LIN {X 0,Y 136.001,Z 403.544,A -85,B 0,C 180,E1 -24793.658,E2 -24793.658} C_VEL
LIN {X 0,Y 136.034,Z 403.535,A -85,B 0,C 180,E1 -24797.807,E2 -24797.807} C_VEL
LIN {X 0,Y 136.073,Z 403.535,A -85,B 0,C 180,E1 -24801.699,E2 -24801.699} C_VEL
LIN {X 0,Y 136.278,Z 403.501,A -85,B 0,C 180,E1 -24805.603,E2 -24805.603} C_VEL
LIN {X 0,Y 136.386,Z 403.498,A -85,B 0,C 180,E1 -24808.982,E2 -24808.982} C_VEL
LIN {X 0,Y 136.062,Z 403.665,A -85,B 0,C 180,E1 -24810.402,E2 -24810.402} C_VEL
LIN {X 0,Y 135.119,Z 409.074,A -85,B 0,C 180,E1 -24817.039,E2 -24817.039} C_VEL
LIN {X 0,Y 134.458,Z 414.255,A -85,B 0,C 180,E1 -24823.293,E2 -24823.293} C_VEL
LIN {X 0,Y 135.285,Z 420.732,A -85,B 0,C 180,E1 -24831.034,E2 -24831.034} C_VEL
LIN {X 0,Y 135.533,Z 421.149,A -85,B 0,C 180,E1 -24831.52,E2 -24831.52} C_VEL
LIN {X 0,Y 136.845,Z 432.369,A -85,B 0,C 180,E1 -24833.364,E2 -24833.364} C_VEL
LIN {X 0,Y 136.477,Z 444.992,A -85,B 0,C 180,E1 -24836.309,E2 -24836.309} C_VEL
LIN {X 0,Y 136.219,Z 455.03,A -85,B 0,C 180,E1 -24839.261,E2 -24839.261} C_VEL
LIN {X 0,Y 136.014,Z 464.96,A -85,B 0,C 180,E1 -24842.962,E2 -24842.962} C_VEL
LIN {X 0,Y 136.62,Z 474.818,A -85,B 0,C 180,E1 -24847.389,E2 -24847.389} C_VEL
LIN {X 0,Y 138.11,Z 482.79,A -85,B 0,C 180,E1 -24851.744,E2 -24851.744} C_VEL
LIN {X 0,Y 140.744,Z 489.39,A -85,B 0,C 180,E1 -24855.941,E2 -24855.941} C_VEL
LIN {X 0,Y 144.372,Z 494.762,A -85,B 0,C 180,E1 -24859.923,E2 -24859.923} C_VEL
LIN {X 0,Y 148.92,Z 499.026,A -85,B 0,C 180,E1 -24863.65,E2 -24863.65} C_VEL
LIN {X 0,Y 154.307,Z 502.234,A -85,B 0,C 180,E1 -24867.094,E2 -24867.094} C_VEL
LIN {X 0,Y 158.302,Z 503.827,A -85,B 0,C 180,E1 -24869.233,E2 -24869.233} C_VEL
LIN {X 0,Y 162.598,Z 504.999,A -85,B 0,C 180,E1 -24871.244,E2 -24871.244} C_VEL
LIN {X 0,Y 169.94,Z 505.976,A -85,B 0,C 180,E1 -24874.196,E2 -24874.196} C_VEL
LIN {X 0,Y 171.965,Z 506.075,A -85,B 0,C 180,E1 -24874.901,E2 -24874.901} C_VEL
LIN {X 0,Y 176.179,Z 506.156,A -85,B 0,C 180,E1 -24876.753,E2 -24876.753} C_VEL
LIN {X 0,Y 178.352,Z 506.601,A -85,B 0,C 180,E1 -24879.086,E2 -24879.086} C_VEL
LIN {X 0,Y 180.016,Z 507.386,A -85,B 0,C 180,E1 -24882.116,E2 -24882.116} C_VEL
LIN {X 0,Y 179.621,Z 508.08,A -85,B 0,C 180,E1 -24883.626,E2 -24883.626} C_VEL
LIN {X 0,Y 177.585,Z 508.851,A -85,B 0,C 180,E1 -24884.572,E2 -24884.572} C_VEL
LIN {X 0,Y 167.712,Z 511.361,A -85,B 0,C 180,E1 -24887.895,E2 -24887.895} C_VEL
LIN {X 0,Y 163.054,Z 512.165,A -85,B 0,C 180,E1 -24889.718,E2 -24889.718} C_VEL
LIN {X 0,Y 154.89,Z 513.005,A -85,B 0,C 180,E1 -24893.852,E2 -24893.852} C_VEL
LIN {X 0,Y 147.172,Z 512.738,A -85,B 0,C 180,E1 -24899.268,E2 -24899.268} C_VEL
LIN {X 0,Y 142.861,Z 511.656,A -85,B 0,C 180,E1 -24903.72,E2 -24903.72} C_VEL
LIN {X 0,Y 139.41,Z 509.457,A -85,B 0,C 180,E1 -24909.335,E2 -24909.335} C_VEL
LIN {X 0,Y 137.831,Z 505.899,A -85,B 0,C 180,E1 -24915.653,E2 -24915.653} C_VEL
LIN {X 0,Y 138.323,Z 501.685,A -85,B 0,C 180,E1 -24921.232,E2 -24921.232} C_VEL
LIN {X 0,Y 139.606,Z 497.302,A -85,B 0,C 180,E1 -24925.669,E2 -24925.669} C_VEL
LIN {X 0,Y 140.175,Z 494.465,A -85,B 0,C 180,E1 -24927.844,E2 -24927.844} C_VEL
LIN {X 0,Y 140.099,Z 489.468,A -85,B 0,C 180,E1 -24930.718,E2 -24930.718} C_VEL
LIN {X 0,Y 139.615,Z 481.506,A -85,B 0,C 180,E1 -24934.33,E2 -24934.33} C_VEL
LIN {X 0,Y 139.3,Z 472.487,A -85,B 0,C 180,E1 -24937.61,E2 -24937.61} C_VEL
LIN {X 0,Y 139.429,Z 464.069,A -85,B 0,C 180,E1 -24940.161,E2 -24940.161} C_VEL
LIN {X 0,Y 137.814,Z 452.885,A -85,B 0,C 180,E1 -24942.565,E2 -24942.565} C_VEL
LIN {X 0,Y 136.785,Z 440.476,A -85,B 0,C 180,E1 -24944.679,E2 -24944.679} C_VEL
LIN {X 0,Y 136.596,Z 432.577,A -85,B 0,C 180,E1 -24945.766,E2 -24945.766} C_VEL
LIN {X 0,Y 136.082,Z 427.218,A -85,B 0,C 180,E1 -24951.193,E2 -24951.193} C_VEL
LIN {X 0,Y 138.905,Z 417.791,A -85,B 0,C 180,E1 -24960.669,E2 -24960.669} C_VEL
LIN {X 0,Y 139.445,Z 416.478,A -85,B 0,C 180,E1 -24961.949,E2 -24961.949} C_VEL
LIN {X 0,Y 138.943,Z 413.586,A -85,B 0,C 180,E1 -24964.73,E2 -24964.73} C_VEL
LIN {X 0,Y 137.461,Z 408.348,A -85,B 0,C 180,E1 -24969.923,E2 -24969.923} C_VEL
LIN {X 0,Y 136.332,Z 403.499,A -85,B 0,C 180,E1 -24975.017,E2 -24975.017} C_VEL
LIN {X 0,Y 136.064,Z 403.536,A -85,B 0,C 180,E1 -24981.697,E2 -24981.697} C_VEL
LIN {X 0,Y 136.09,Z 403.527,A -85,B 0,C 180,E1 -24985.717,E2 -24985.717} C_VEL
LIN {X 0,Y 136.146,Z 403.523,A -85,B 0,C 180,E1 -24992.316,E2 -24992.316} C_VEL
LIN {X 0,Y 136.19,Z 403.52,A -85,B 0,C 180,E1 -24998.168,E2 -24998.168} C_VEL
LIN {X 0,Y 135.722,Z 403.592,A -85,B 0,C 180,E1 -25000.636,E2 -25000.636} C_VEL
LIN {X 0,Y 134.282,Z 403.775,A -85,B 0,C 180,E1 -25003.077,E2 -25003.077} C_VEL
LIN {X 0,Y 129.836,Z 404.308,A -85,B 0,C 180,E1 -25009.8,E2 -25009.8} C_VEL
LIN {X 0,Y 129.486,Z 404.346,A -85,B 0,C 180,E1 -25011.576,E2 -25011.576} C_VEL
LIN {X 0,Y 130.091,Z 404.274,A -85,B 0,C 180,E1 -25020,E2 -25020} C_VEL
LIN {X 0,Y 129.531,Z 404.344,A -85,B 0,C 180,E1 -25029.368,E2 -25029.368} C_VEL
LIN {X 0,Y 129.395,Z 404.366,A -85,B 0,C 180,E1 -25032.548,E2 -25032.548} C_VEL
LIN {X 0,Y 129.164,Z 404.393,A -85,B 0,C 180,E1 -25039.055,E2 -25039.055} C_VEL
LIN {X 0,Y 129.109,Z 404.402,A -85,B 0,C 180,E1 -25042.398,E2 -25042.398} C_VEL
LIN {X 0,Y 129.036,Z 404.412,A -85,B 0,C 180,E1 -25049.374,E2 -25049.374} C_VEL
LIN {X 0,Y 128.961,Z 404.416,A -85,B 0,C 180,E1 -25055.17,E2 -25055.17} C_VEL
LIN {X 0,Y 128.934,Z 404.422,A -85,B 0,C 180,E1 -25060.852,E2 -25060.852} C_VEL
LIN {X 0,Y 128.922,Z 404.425,A -85,B 0,C 180,E1 -25065.128,E2 -25065.128} C_VEL
LIN {X 0,Y 128.958,Z 404.418,A -85,B 0,C 180,E1 -25069.728,E2 -25069.728} C_VEL
LIN {X 0,Y 128.993,Z 404.418,A -85,B 0,C 180,E1 -25074.811,E2 -25074.811} C_VEL
LIN {X 0,Y 129.034,Z 404.406,A -85,B 0,C 180,E1 -25080.647,E2 -25080.647} C_VEL
LIN {X 0,Y 129.137,Z 404.395,A -85,B 0,C 180,E1 -25087.607,E2 -25087.607} C_VEL
LIN {X 0,Y 129.188,Z 404.391,A -85,B 0,C 180,E1 -25090.95,E2 -25090.95} C_VEL
LIN {X 0,Y 129.418,Z 404.357,A -85,B 0,C 180,E1 -25097.821,E2 -25097.821} C_VEL
LIN {X 0,Y 129.519,Z 404.351,A -85,B 0,C 180,E1 -25100.632,E2 -25100.632} C_VEL
LIN {X 0,Y 130.092,Z 404.281,A -85,B 0,C 180,E1 -25110.001,E2 -25110.001} C_VEL
LIN {X 0,Y 129.479,Z 404.356,A -85,B 0,C 180,E1 -25119.372,E2 -25119.372} C_VEL
LIN {X 0,Y 129.347,Z 404.365,A -85,B 0,C 180,E1 -25122.553,E2 -25122.553} C_VEL
LIN {X 0,Y 129.159,Z 404.395,A -85,B 0,C 180,E1 -25129.056,E2 -25129.056} C_VEL
LIN {X 0,Y 129.111,Z 404.398,A -85,B 0,C 180,E1 -25132.399,E2 -25132.399} C_VEL
LIN {X 0,Y 129.038,Z 404.406,A -85,B 0,C 180,E1 -25139.374,E2 -25139.374} C_VEL
LIN {X 0,Y 128.995,Z 404.418,A -85,B 0,C 180,E1 -25145.19,E2 -25145.19} C_VEL
LIN {X 0,Y 128.953,Z 404.419,A -85,B 0,C 180,E1 -25150.845,E2 -25150.845} C_VEL
LIN {X 0,Y 128.924,Z 404.423,A -85,B 0,C 180,E1 -25155.128,E2 -25155.128} C_VEL
LIN {X 0,Y 128.987,Z 404.417,A -85,B 0,C 180,E1 -25159.713,E2 -25159.713} C_VEL
LIN {X 0,Y 129.144,Z 404.393,A -85,B 0,C 180,E1 -25164.717,E2 -25164.717} C_VEL
LIN {X 0,Y 129.235,Z 404.374,A -85,B 0,C 180,E1 -25167.056,E2 -25167.056} C_VEL
LIN {X 0,Y 128.884,Z 404.599,A -85,B 0,C 180,E1 -25171.009,E2 -25171.009} C_VEL
LIN {X 0,Y 127.961,Z 409.6,A -85,B 0,C 180,E1 -25177.39,E2 -25177.39} C_VEL
LIN {X 0,Y 127.313,Z 414.748,A -85,B 0,C 180,E1 -25183.977,E2 -25183.977} C_VEL
LIN {X 0,Y 128.098,Z 420.318,A -85,B 0,C 180,E1 -25190.957,E2 -25190.957} C_VEL
LIN {X 0,Y 128.762,Z 421.528,A -85,B 0,C 180,E1 -25192.435,E2 -25192.435} C_VEL
LIN {X 0,Y 130.011,Z 431.845,A -85,B 0,C 180,E1 -25194.183,E2 -25194.183} C_VEL
LIN {X 0,Y 129.718,Z 443.147,A -85,B 0,C 180,E1 -25196.894,E2 -25196.894} C_VEL
LIN {X 0,Y 129.538,Z 453.363,A -85,B 0,C 180,E1 -25200,E2 -25200} C_VEL
LIN {X 0,Y 129.381,Z 463.671,A -85,B 0,C 180,E1 -25203.893,E2 -25203.893} C_VEL
LIN {X 0,Y 129.901,Z 472.26,A -85,B 0,C 180,E1 -25207.773,E2 -25207.773} C_VEL
LIN {X 0,Y 131.762,Z 482.01,A -85,B 0,C 180,E1 -25213.102,E2 -25213.102} C_VEL
LIN {X 0,Y 134.607,Z 488.854,A -85,B 0,C 180,E1 -25217.47,E2 -25217.47} C_VEL
LIN {X 0,Y 139.21,Z 495.266,A -85,B 0,C 180,E1 -25222.249,E2 -25222.249} C_VEL
LIN {X 0,Y 144.183,Z 499.613,A -85,B 0,C 180,E1 -25226.021,E2 -25226.021} C_VEL
LIN {X 0,Y 147.992,Z 501.924,A -85,B 0,C 180,E1 -25228.352,E2 -25228.352} C_VEL
LIN {X 0,Y 152.112,Z 503.822,A -85,B 0,C 180,E1 -25230.546,E2 -25230.546} C_VEL
LIN {X 0,Y 156.554,Z 505.286,A -85,B 0,C 180,E1 -25232.595,E2 -25232.595} C_VEL
LIN {X 0,Y 164.524,Z 506.798,A -85,B 0,C 180,E1 -25235.744,E2 -25235.744} C_VEL
LIN {X 0,Y 166.167,Z 506.978,A -85,B 0,C 180,E1 -25236.308,E2 -25236.308} C_VEL
LIN {X 0,Y 170.317,Z 507.393,A -85,B 0,C 180,E1 -25238.241,E2 -25238.241} C_VEL
LIN {X 0,Y 172.203,Z 508.123,A -85,B 0,C 180,E1 -25240.768,E2 -25240.768} C_VEL
LIN {X 0,Y 172.597,Z 508.889,A -85,B 0,C 180,E1 -25242.865,E2 -25242.865} C_VEL
LIN {X 0,Y 162.539,Z 510.833,A -85,B 0,C 180,E1 -25246.225,E2 -25246.225} C_VEL
LIN {X 0,Y 157.737,Z 511.376,A -85,B 0,C 180,E1 -25248.061,E2 -25248.061} C_VEL
LIN {X 0,Y 149.294,Z 511.755,A -85,B 0,C 180,E1 -25252.267,E2 -25252.267} C_VEL
LIN {X 0,Y 141.83,Z 511.081,A -85,B 0,C 180,E1 -25257.394,E2 -25257.394} C_VEL
LIN {X 0,Y 136.776,Z 509.594,A -85,B 0,C 180,E1 -25262.454,E2 -25262.454} C_VEL
LIN {X 0,Y 133.152,Z 507.034,A -85,B 0,C 180,E1 -25268.316,E2 -25268.316} C_VEL
LIN {X 0,Y 131.562,Z 503.393,A -85,B 0,C 180,E1 -25274.508,E2 -25274.508} C_VEL
LIN {X 0,Y 131.998,Z 498.616,A -85,B 0,C 180,E1 -25280.808,E2 -25280.808} C_VEL
LIN {X 0,Y 133.399,Z 493.899,A -85,B 0,C 180,E1 -25285.468,E2 -25285.468} C_VEL
LIN {X 0,Y 133.899,Z 490.875,A -85,B 0,C 180,E1 -25287.743,E2 -25287.743} C_VEL
LIN {X 0,Y 133.538,Z 485.851,A -85,B 0,C 180,E1 -25290.525,E2 -25290.525} C_VEL
LIN {X 0,Y 133.112,Z 478.587,A -85,B 0,C 180,E1 -25293.784,E2 -25293.784} C_VEL
LIN {X 0,Y 132.773,Z 469.166,A -85,B 0,C 180,E1 -25297.221,E2 -25297.221} C_VEL
LIN {X 0,Y 132.831,Z 462.944,A -85,B 0,C 180,E1 -25299.133,E2 -25299.133} C_VEL
LIN {X 0,Y 131.036,Z 450.859,A -85,B 0,C 180,E1 -25301.799,E2 -25301.799} C_VEL
LIN {X 0,Y 130.027,Z 438.226,A -85,B 0,C 180,E1 -25304.003,E2 -25304.003} C_VEL
LIN {X 0,Y 129.763,Z 432.188,A -85,B 0,C 180,E1 -25304.932,E2 -25304.932} C_VEL
LIN {X 0,Y 128.957,Z 428.337,A -85,B 0,C 180,E1 -25309.086,E2 -25309.086} C_VEL
LIN {X 0,Y 132.142,Z 416.641,A -85,B 0,C 180,E1 -25321.683,E2 -25321.683} C_VEL
LIN {X 0,Y 132.309,Z 416.249,A -85,B 0,C 180,E1 -25322.085,E2 -25322.085} C_VEL
LIN {X 0,Y 131.69,Z 413.387,A -85,B 0,C 180,E1 -25325.008,E2 -25325.008} C_VEL
LIN {X 0,Y 130.12,Z 407.807,A -85,B 0,C 180,E1 -25330.872,E2 -25330.872} C_VEL
LIN {X 0,Y 129.313,Z 404.374,A -85,B 0,C 180,E1 -25334.799,E2 -25334.799} C_VEL
LIN {X 0,Y 129.005,Z 404.414,A -85,B 0,C 180,E1 -25339.702,E2 -25339.702} C_VEL
LIN {X 0,Y 128.993,Z 404.411,A -85,B 0,C 180,E1 -25344.81,E2 -25344.81} C_VEL
LIN {X 0,Y 129.033,Z 404.411,A -85,B 0,C 180,E1 -25350.646,E2 -25350.646} C_VEL
LIN {X 0,Y 129.108,Z 404.402,A -85,B 0,C 180,E1 -25357.602,E2 -25357.602} C_VEL
LIN {X 0,Y 129.16,Z 404.394,A -85,B 0,C 180,E1 -25360.945,E2 -25360.945} C_VEL
LIN {X 0,Y 129.419,Z 404.364,A -85,B 0,C 180,E1 -25367.815,E2 -25367.815} C_VEL
LIN {X 0,Y 129.486,Z 404.346,A -85,B 0,C 180,E1 -25371.576,E2 -25371.576} C_VEL
LIN {X 0,Y 128.783,Z 404.442,A -85,B 0,C 180,E1 -25374.182,E2 -25374.182} C_VEL
LIN {X 0,Y 127.224,Z 404.637,A -85,B 0,C 180,E1 -25376.756,E2 -25376.756} C_VEL
LIN {X 0,Y 122.783,Z 405.191,A -85,B 0,C 180,E1 -25383.868,E2 -25383.868} C_VEL
LIN {X 0,Y 122.457,Z 405.224,A -85,B 0,C 180,E1 -25385.748,E2 -25385.748} C_VEL
LIN {X 0,Y 122.457,Z 405.228,A -85,B 0,C 180,E1 -25389.914,E2 -25389.914} C_VEL
LIN {X 0,Y 122.287,Z 405.253,A -85,B 0,C 180,E1 -25393.29,E2 -25393.29} C_VEL
LIN {X 0,Y 122.052,Z 405.28,A -85,B 0,C 180,E1 -25400.212,E2 -25400.212} C_VEL
LIN {X 0,Y 121.984,Z 405.287,A -85,B 0,C 180,E1 -25403.785,E2 -25403.785} C_VEL
LIN {X 0,Y 121.939,Z 405.295,A -85,B 0,C 180,E1 -25410.172,E2 -25410.172} C_VEL
LIN {X 0,Y 121.886,Z 405.299,A -85,B 0,C 180,E1 -25416.173,E2 -25416.173} C_VEL
LIN {X 0,Y 121.873,Z 405.299,A -85,B 0,C 180,E1 -25421.439,E2 -25421.439} C_VEL
LIN {X 0,Y 121.885,Z 405.302,A -85,B 0,C 180,E1 -25428.556,E2 -25428.556} C_VEL
LIN {X 0,Y 121.946,Z 405.296,A -85,B 0,C 180,E1 -25434.809,E2 -25434.809} C_VEL
LIN {X 0,Y 121.943,Z 405.289,A -85,B 0,C 180,E1 -25439.827,E2 -25439.827} C_VEL
LIN {X 0,Y 122.069,Z 405.275,A -85,B 0,C 180,E1 -25447.1,E2 -25447.1} C_VEL
LIN {X 0,Y 122.133,Z 405.271,A -85,B 0,C 180,E1 -25453.279,E2 -25453.279} C_VEL
LIN {X 0,Y 122.365,Z 405.235,A -85,B 0,C 180,E1 -25457.527,E2 -25457.527} C_VEL
LIN {X 0,Y 122.448,Z 405.231,A -85,B 0,C 180,E1 -25460.086,E2 -25460.086} C_VEL
LIN {X 0,Y 122.608,Z 405.208,A -85,B 0,C 180,E1 -25466.715,E2 -25466.715} C_VEL
LIN {X 0,Y 123.045,Z 405.159,A -85,B 0,C 180,E1 -25470.001,E2 -25470.001} C_VEL
LIN {X 0,Y 122.428,Z 405.233,A -85,B 0,C 180,E1 -25476.593,E2 -25476.593} C_VEL
LIN {X 0,Y 122.32,Z 405.241,A -85,B 0,C 180,E1 -25482.377,E2 -25482.377} C_VEL
LIN {X 0,Y 122.114,Z 405.273,A -85,B 0,C 180,E1 -25486.725,E2 -25486.725} C_VEL
LIN {X 0,Y 122.026,Z 405.28,A -85,B 0,C 180,E1 -25492.852,E2 -25492.852} C_VEL
LIN {X 0,Y 121.952,Z 405.293,A -85,B 0,C 180,E1 -25497.455,E2 -25497.455} C_VEL
LIN {X 0,Y 121.914,Z 405.294,A -85,B 0,C 180,E1 -25501.254,E2 -25501.254} C_VEL
LIN {X 0,Y 121.914,Z 405.296,A -85,B 0,C 180,E1 -25506.19,E2 -25506.19} C_VEL
LIN {X 0,Y 121.886,Z 405.302,A -85,B 0,C 180,E1 -25511.445,E2 -25511.445} C_VEL
LIN {X 0,Y 121.905,Z 405.295,A -85,B 0,C 180,E1 -25518.545,E2 -25518.545} C_VEL
LIN {X 0,Y 122.098,Z 405.27,A -85,B 0,C 180,E1 -25524.858,E2 -25524.858} C_VEL
LIN {X 0,Y 121.921,Z 405.299,A -85,B 0,C 180,E1 -25529.846,E2 -25529.846} C_VEL
LIN {X 0,Y 121.709,Z 405.375,A -85,B 0,C 180,E1 -25531.483,E2 -25531.483} C_VEL
LIN {X 0,Y 120.729,Z 410.686,A -85,B 0,C 180,E1 -25538.657,E2 -25538.657} C_VEL
LIN {X 0,Y 120.948,Z 419.961,A -85,B 0,C 180,E1 -25551.057,E2 -25551.057} C_VEL
LIN {X 0,Y 122.082,Z 421.848,A -85,B 0,C 180,E1 -25553.492,E2 -25553.492} C_VEL
LIN {X 0,Y 123.242,Z 430.964,A -85,B 0,C 180,E1 -25555.093,E2 -25555.093} C_VEL
LIN {X 0,Y 123.053,Z 442.392,A -85,B 0,C 180,E1 -25557.954,E2 -25557.954} C_VEL
LIN {X 0,Y 122.867,Z 452.781,A -85,B 0,C 180,E1 -25561.229,E2 -25561.229} C_VEL
LIN {X 0,Y 122.826,Z 462.229,A -85,B 0,C 180,E1 -25564.924,E2 -25564.924} C_VEL
LIN {X 0,Y 123.665,Z 472.552,A -85,B 0,C 180,E1 -25569.816,E2 -25569.816} C_VEL
LIN {X 0,Y 125.507,Z 481.087,A -85,B 0,C 180,E1 -25574.595,E2 -25574.595} C_VEL
LIN {X 0,Y 129.23,Z 489.194,A -85,B 0,C 180,E1 -25579.871,E2 -25579.871} C_VEL
LIN {X 0,Y 134.352,Z 495.717,A -85,B 0,C 180,E1 -25584.739,E2 -25584.739} C_VEL
LIN {X 0,Y 139.769,Z 500.125,A -85,B 0,C 180,E1 -25588.535,E2 -25588.535} C_VEL
LIN {X 0,Y 146.012,Z 503.562,A -85,B 0,C 180,E1 -25591.969,E2 -25591.969} C_VEL
LIN {X 0,Y 150.591,Z 505.329,A -85,B 0,C 180,E1 -25594.058,E2 -25594.058} C_VEL
LIN {X 0,Y 160.467,Z 507.634,A -85,B 0,C 180,E1 -25597.818,E2 -25597.818} C_VEL
LIN {X 0,Y 163.978,Z 508.255,A -85,B 0,C 180,E1 -25599.513,E2 -25599.513} C_VEL
LIN {X 0,Y 165.047,Z 509.13,A -85,B 0,C 180,E1 -25601.96,E2 -25601.96} C_VEL
LIN {X 0,Y 157.519,Z 510.057,A -85,B 0,C 180,E1 -25604.449,E2 -25604.449} C_VEL
LIN {X 0,Y 152.587,Z 510.353,A -85,B 0,C 180,E1 -25606.299,E2 -25606.299} C_VEL
LIN {X 0,Y 143.872,Z 510.261,A -85,B 0,C 180,E1 -25610.576,E2 -25610.576} C_VEL
LIN {X 0,Y 136.512,Z 509.25,A -85,B 0,C 180,E1 -25615.506,E2 -25615.506} C_VEL
LIN {X 0,Y 130.835,Z 507.311,A -85,B 0,C 180,E1 -25621.088,E2 -25621.088} C_VEL
LIN {X 0,Y 127.037,Z 504.383,A -85,B 0,C 180,E1 -25627.215,E2 -25627.215} C_VEL
LIN {X 0,Y 125.329,Z 500.447,A -85,B 0,C 180,E1 -25633.716,E2 -25633.716} C_VEL
LIN {X 0,Y 125.813,Z 495.311,A -85,B 0,C 180,E1 -25640.352,E2 -25640.352} C_VEL
LIN {X 0,Y 127.058,Z 491.022,A -85,B 0,C 180,E1 -25644.652,E2 -25644.652} C_VEL
LIN {X 0,Y 127.628,Z 488.204,A -85,B 0,C 180,E1 -25646.843,E2 -25646.843} C_VEL
LIN {X 0,Y 127.338,Z 484.049,A -85,B 0,C 180,E1 -25649.209,E2 -25649.209} C_VEL
LIN {X 0,Y 126.675,Z 475.476,A -85,B 0,C 180,E1 -25653.18,E2 -25653.18} C_VEL
LIN {X 0,Y 126.291,Z 465.683,A -85,B 0,C 180,E1 -25656.791,E2 -25656.791} C_VEL
LIN {X 0,Y 126.287,Z 461.842,A -85,B 0,C 180,E1 -25657.997,E2 -25657.997} C_VEL
LIN {X 0,Y 124.345,Z 449.6,A -85,B 0,C 180,E1 -25660.79,E2 -25660.79} C_VEL
LIN {X 0,Y 123.338,Z 437.691,A -85,B 0,C 180,E1 -25662.965,E2 -25662.965} C_VEL
LIN {X 0,Y 123.062,Z 431.903,A -85,B 0,C 180,E1 -25663.865,E2 -25663.865} C_VEL
LIN {X 0,Y 121.953,Z 427.904,A -85,B 0,C 180,E1 -25668.478,E2 -25668.478} C_VEL
LIN {X 0,Y 124.516,Z 417.486,A -85,B 0,C 180,E1 -25680.529,E2 -25680.529} C_VEL
LIN {X 0,Y 125.097,Z 415.628,A -85,B 0,C 180,E1 -25682.573,E2 -25682.573} C_VEL
LIN {X 0,Y 124.309,Z 412.645,A -85,B 0,C 180,E1 -25685.829,E2 -25685.829} C_VEL
LIN {X 0,Y 122.775,Z 407.228,A -85,B 0,C 180,E1 -25691.913,E2 -25691.913} C_VEL
LIN {X 0,Y 122.324,Z 405.246,A -85,B 0,C 180,E1 -25694.206,E2 -25694.206} C_VEL
LIN {X 0,Y 121.906,Z 405.3,A -85,B 0,C 180,E1 -25700.642,E2 -25700.642} C_VEL
LIN {X 0,Y 121.946,Z 405.289,A -85,B 0,C 180,E1 -25704.808,E2 -25704.808} C_VEL
LIN {X 0,Y 121.942,Z 405.296,A -85,B 0,C 180,E1 -25709.826,E2 -25709.826} C_VEL
LIN {X 0,Y 121.983,Z 405.288,A -85,B 0,C 180,E1 -25716.215,E2 -25716.215} C_VEL
LIN {X 0,Y 122.05,Z 405.282,A -85,B 0,C 180,E1 -25719.788,E2 -25719.788} C_VEL
LIN {X 0,Y 122.264,Z 405.254,A -85,B 0,C 180,E1 -25726.707,E2 -25726.707} C_VEL
LIN {X 0,Y 122.407,Z 405.227,A -85,B 0,C 180,E1 -25731.567,E2 -25731.567} C_VEL
LIN {X 0,Y 123.045,Z 405.151,A -85,B 0,C 180,E1 -25740,E2 -25740} C_VEL
LIN {X 0,Y 122.457,Z 405.224,A -85,B 0,C 180,E1 -25745.748,E2 -25745.748} C_VEL
LIN {X 0,Y 121.708,Z 405.325,A -85,B 0,C 180,E1 -25748.488,E2 -25748.488} C_VEL
LIN {X 0,Y 120.01,Z 405.539,A -85,B 0,C 180,E1 -25751.186,E2 -25751.186} C_VEL
LIN {X 0,Y 115.236,Z 406.126,A -85,B 0,C 180,E1 -25758.688,E2 -25758.688} C_VEL
LIN {X 0,Y 114.949,Z 406.16,A -85,B 0,C 180,E1 -25760.688,E2 -25760.688} C_VEL
LIN {X 0,Y 114.874,Z 406.169,A -85,B 0,C 180,E1 -25765.357,E2 -25765.357} C_VEL
LIN {X 0,Y 114.862,Z 406.177,A -85,B 0,C 180,E1 -25771.063,E2 -25771.063} C_VEL
LIN {X 0,Y 114.781,Z 406.187,A -85,B 0,C 180,E1 -25777.756,E2 -25777.756} C_VEL
LIN {X 0,Y 114.787,Z 406.18,A -85,B 0,C 180,E1 -25782.718,E2 -25782.718} C_VEL
LIN {X 0,Y 114.803,Z 406.184,A -85,B 0,C 180,E1 -25787.671,E2 -25787.671} C_VEL
LIN {X 0,Y 114.812,Z 406.178,A -85,B 0,C 180,E1 -25792.728,E2 -25792.728} C_VEL
LIN {X 0,Y 114.869,Z 406.17,A -85,B 0,C 180,E1 -25798.932,E2 -25798.932} C_VEL
LIN {X 0,Y 114.967,Z 406.161,A -85,B 0,C 180,E1 -25806.486,E2 -25806.486} C_VEL
LIN {X 0,Y 115.035,Z 406.156,A -85,B 0,C 180,E1 -25812.214,E2 -25812.214} C_VEL
LIN {X 0,Y 115.307,Z 406.114,A -85,B 0,C 180,E1 -25817.216,E2 -25817.216} C_VEL
LIN {X 0,Y 115.391,Z 406.11,A -85,B 0,C 180,E1 -25823.004,E2 -25823.004} C_VEL
LIN {X 0,Y 115.996,Z 406.037,A -85,B 0,C 180,E1 -25830.001,E2 -25830.001} C_VEL
LIN {X 0,Y 115.368,Z 406.112,A -85,B 0,C 180,E1 -25836.999,E2 -25836.999} C_VEL
LIN {X 0,Y 115.254,Z 406.12,A -85,B 0,C 180,E1 -25842.668,E2 -25842.668} C_VEL
LIN {X 0,Y 115.016,Z 406.158,A -85,B 0,C 180,E1 -25847.79,E2 -25847.79} C_VEL
LIN {X 0,Y 114.949,Z 406.163,A -85,B 0,C 180,E1 -25853.493,E2 -25853.493} C_VEL
LIN {X 0,Y 114.871,Z 406.17,A -85,B 0,C 180,E1 -25861.069,E2 -25861.069} C_VEL
LIN {X 0,Y 114.804,Z 406.178,A -85,B 0,C 180,E1 -25867.748,E2 -25867.748} C_VEL
LIN {X 0,Y 114.797,Z 406.185,A -85,B 0,C 180,E1 -25872.722,E2 -25872.722} C_VEL
LIN {X 0,Y 114.818,Z 406.177,A -85,B 0,C 180,E1 -25877.677,E2 -25877.677} C_VEL
LIN {X 0,Y 114.913,Z 406.171,A -85,B 0,C 180,E1 -25882.663,E2 -25882.663} C_VEL
LIN {X 0,Y 114.937,Z 406.168,A -85,B 0,C 180,E1 -25888.877,E2 -25888.877} C_VEL
LIN {X 0,Y 114.436,Z 406.321,A -85,B 0,C 180,E1 -25892.325,E2 -25892.325} C_VEL
LIN {X 0,Y 113.662,Z 410.469,A -85,B 0,C 180,E1 -25898.223,E2 -25898.223} C_VEL
LIN {X 0,Y 113.817,Z 419.533,A -85,B 0,C 180,E1 -25911.109,E2 -25911.109} C_VEL
LIN {X 0,Y 115.466,Z 422.251,A -85,B 0,C 180,E1 -25914.762,E2 -25914.762} C_VEL
LIN {X 0,Y 116.575,Z 431.74,A -85,B 0,C 180,E1 -25916.544,E2 -25916.544} C_VEL
LIN {X 0,Y 116.415,Z 443.035,A -85,B 0,C 180,E1 -25919.568,E2 -25919.568} C_VEL
LIN {X 0,Y 116.315,Z 451.979,A -85,B 0,C 180,E1 -25922.597,E2 -25922.597} C_VEL
LIN {X 0,Y 116.473,Z 462.434,A -85,B 0,C 180,E1 -25926.931,E2 -25926.931} C_VEL
LIN {X 0,Y 117.576,Z 472.798,A -85,B 0,C 180,E1 -25932.076,E2 -25932.076} C_VEL
LIN {X 0,Y 120.369,Z 482.53,A -85,B 0,C 180,E1 -25937.85,E2 -25937.85} C_VEL
LIN {X 0,Y 124.125,Z 489.494,A -85,B 0,C 180,E1 -25942.469,E2 -25942.469} C_VEL
LIN {X 0,Y 129.793,Z 496.076,A -85,B 0,C 180,E1 -25947.404,E2 -25947.404} C_VEL
LIN {X 0,Y 135.634,Z 500.59,A -85,B 0,C 180,E1 -25951.209,E2 -25951.209} C_VEL
LIN {X 0,Y 144.719,Z 505.131,A -85,B 0,C 180,E1 -25955.645,E2 -25955.645} C_VEL
LIN {X 0,Y 154.876,Z 508.025,A -85,B 0,C 180,E1 -25959.442,E2 -25959.442} C_VEL
LIN {X 0,Y 157.371,Z 508.605,A -85,B 0,C 180,E1 -25960.605,E2 -25960.605} C_VEL
LIN {X 0,Y 152.685,Z 509.027,A -85,B 0,C 180,E1 -25962.567,E2 -25962.567} C_VEL
LIN {X 0,Y 142.99,Z 508.929,A -85,B 0,C 180,E1 -25966.519,E2 -25966.519} C_VEL
LIN {X 0,Y 134.592,Z 507.929,A -85,B 0,C 180,E1 -25971.199,E2 -25971.199} C_VEL
LIN {X 0,Y 127.773,Z 506.08,A -85,B 0,C 180,E1 -25976.63,E2 -25976.63} C_VEL
LIN {X 0,Y 122.803,Z 503.302,A -85,B 0,C 180,E1 -25982.752,E2 -25982.752} C_VEL
LIN {X 0,Y 119.75,Z 499.201,A -85,B 0,C 180,E1 -25989.889,E2 -25989.889} C_VEL
LIN {X 0,Y 119.198,Z 494.693,A -85,B 0,C 180,E1 -25996.358,E2 -25996.358} C_VEL
LIN {X 0,Y 120.693,Z 488.468,A -85,B 0,C 180,E1 -26003.311,E2 -26003.311} C_VEL
LIN {X 0,Y 121.302,Z 486.05,A -85,B 0,C 180,E1 -26005.411,E2 -26005.411} C_VEL
LIN {X 0,Y 121.34,Z 483.092,A -85,B 0,C 180,E1 -26007.302,E2 -26007.302} C_VEL
LIN {X 0,Y 120.476,Z 474.068,A -85,B 0,C 180,E1 -26011.672,E2 -26011.672} C_VEL
LIN {X 0,Y 119.931,Z 464.125,A -85,B 0,C 180,E1 -26015.504,E2 -26015.504} C_VEL
LIN {X 0,Y 119.838,Z 460.392,A -85,B 0,C 180,E1 -26016.735,E2 -26016.735} C_VEL
LIN {X 0,Y 117.735,Z 447.974,A -85,B 0,C 180,E1 -26019.664,E2 -26019.664} C_VEL
LIN {X 0,Y 116.574,Z 434.552,A -85,B 0,C 180,E1 -26022.181,E2 -26022.181} C_VEL
LIN {X 0,Y 116.455,Z 431.627,A -85,B 0,C 180,E1 -26022.636,E2 -26022.636} C_VEL
LIN {X 0,Y 115.22,Z 428.871,A -85,B 0,C 180,E1 -26025.931,E2 -26025.931} C_VEL
LIN {X 0,Y 117.362,Z 417.106,A -85,B 0,C 180,E1 -26040.597,E2 -26040.597} C_VEL
LIN {X 0,Y 117.916,Z 415.553,A -85,B 0,C 180,E1 -26042.439,E2 -26042.439} C_VEL
LIN {X 0,Y 116.843,Z 411.674,A -85,B 0,C 180,E1 -26046.976,E2 -26046.976} C_VEL
LIN {X 0,Y 115.308,Z 406.121,A -85,B 0,C 180,E1 -26053.893,E2 -26053.893} C_VEL
LIN {X 0,Y 114.826,Z 406.18,A -85,B 0,C 180,E1 -26062.718,E2 -26062.718} C_VEL
LIN {X 0,Y 114.869,Z 406.176,A -85,B 0,C 180,E1 -26068.932,E2 -26068.932} C_VEL
LIN {X 0,Y 114.947,Z 406.165,A -85,B 0,C 180,E1 -26076.507,E2 -26076.507} C_VEL
LIN {X 0,Y 115.019,Z 406.15,A -85,B 0,C 180,E1 -26082.211,E2 -26082.211} C_VEL
LIN {X 0,Y 115.286,Z 406.124,A -85,B 0,C 180,E1 -26087.257,E2 -26087.257} C_VEL
LIN {X 0,Y 115.393,Z 406.108,A -85,B 0,C 180,E1 -26089.472,E2 -26089.472} C_VEL
LIN {X 0,Y 115.539,Z 406.092,A -85,B 0,C 180,E1 -26096.513,E2 -26096.513} C_VEL
LIN {X 0,Y 115.997,Z 406.029,A -85,B 0,C 180,E1 -26100,E2 -26100} C_VEL
LIN {X 0,Y 115.392,Z 406.107,A -85,B 0,C 180,E1 -26107.104,E2 -26107.104} C_VEL
LIN {X 0,Y 115.287,Z 406.124,A -85,B 0,C 180,E1 -26112.743,E2 -26112.743} C_VEL
LIN {X 0,Y 115.021,Z 406.152,A -85,B 0,C 180,E1 -26117.789,E2 -26117.789} C_VEL
LIN {X 0,Y 114.949,Z 406.16,A -85,B 0,C 180,E1 -26120.688,E2 -26120.688} C_VEL
LIN {X 0,Y 114.328,Z 406.251,A -85,B 0,C 180,E1 -26123.611,E2 -26123.611} C_VEL
LIN {X 0,Y 112.751,Z 406.452,A -85,B 0,C 180,E1 -26126.499,E2 -26126.499} C_VEL
LIN {X 0,Y 108.058,Z 407.023,A -85,B 0,C 180,E1 -26134.528,E2 -26134.528} C_VEL
LIN {X 0,Y 107.688,Z 407.066,A -85,B 0,C 180,E1 -26136.669,E2 -26136.669} C_VEL
LIN {X 0,Y 107.681,Z 407.069,A -85,B 0,C 180,E1 -26140.743,E2 -26140.743} C_VEL
LIN {X 0,Y 107.682,Z 407.07,A -85,B 0,C 180,E1 -26145.884,E2 -26145.884} C_VEL
LIN {X 0,Y 107.707,Z 407.061,A -85,B 0,C 180,E1 -26151.537,E2 -26151.537} C_VEL
LIN {X 0,Y 107.808,Z 407.051,A -85,B 0,C 180,E1 -26158.566,E2 -26158.566} C_VEL
LIN {X 0,Y 107.933,Z 407.036,A -85,B 0,C 180,E1 -26167.003,E2 -26167.003} C_VEL
LIN {X 0,Y 108.053,Z 407.023,A -85,B 0,C 180,E1 -26174.921,E2 -26174.921} C_VEL
LIN {X 0,Y 108.297,Z 406.992,A -85,B 0,C 180,E1 -26178.774,E2 -26178.774} C_VEL
LIN {X 0,Y 108.459,Z 406.968,A -85,B 0,C 180,E1 -26186.285,E2 -26186.285} C_VEL
LIN {X 0,Y 108.946,Z 406.915,A -85,B 0,C 180,E1 -26190.001,E2 -26190.001} C_VEL
LIN {X 0,Y 108.307,Z 406.993,A -85,B 0,C 180,E1 -26197.458,E2 -26197.458} C_VEL
LIN {X 0,Y 108.175,Z 407.002,A -85,B 0,C 180,E1 -26202.957,E2 -26202.957} C_VEL
LIN {X 0,Y 107.908,Z 407.042,A -85,B 0,C 180,E1 -26209.006,E2 -26209.006} C_VEL
LIN {X 0,Y 107.86,Z 407.049,A -85,B 0,C 180,E1 -26214.185,E2 -26214.185} C_VEL
LIN {X 0,Y 107.797,Z 407.056,A -85,B 0,C 180,E1 -26222.052,E2 -26222.052} C_VEL
LIN {X 0,Y 107.709,Z 407.06,A -85,B 0,C 180,E1 -26228.464,E2 -26228.464} C_VEL
LIN {X 0,Y 107.693,Z 407.065,A -85,B 0,C 180,E1 -26235.879,E2 -26235.879} C_VEL
LIN {X 0,Y 107.782,Z 407.059,A -85,B 0,C 180,E1 -26241.489,E2 -26241.489} C_VEL
LIN {X 0,Y 107.874,Z 407.036,A -85,B 0,C 180,E1 -26247.883,E2 -26247.883} C_VEL
LIN {X 0,Y 107.18,Z 407.206,A -85,B 0,C 180,E1 -26253.204,E2 -26253.204} C_VEL
LIN {X 0,Y 106.468,Z 411.029,A -85,B 0,C 180,E1 -26258.993,E2 -26258.993} C_VEL
LIN {X 0,Y 107.106,Z 419.946,A -85,B 0,C 180,E1 -26272.459,E2 -26272.459} C_VEL
LIN {X 0,Y 108.935,Z 422.623,A -85,B 0,C 180,E1 -26276.185,E2 -26276.185} C_VEL
LIN {X 0,Y 109.997,Z 430.534,A -85,B 0,C 180,E1 -26277.711,E2 -26277.711} C_VEL
LIN {X 0,Y 109.952,Z 443.311,A -85,B 0,C 180,E1 -26281.373,E2 -26281.373} C_VEL
LIN {X 0,Y 109.854,Z 453.235,A -85,B 0,C 180,E1 -26285.047,E2 -26285.047} C_VEL
LIN {X 0,Y 110.239,Z 462.606,A -85,B 0,C 180,E1 -26289.171,E2 -26289.171} C_VEL
LIN {X 0,Y 111.729,Z 472.78,A -85,B 0,C 180,E1 -26294.573,E2 -26294.573} C_VEL
LIN {X 0,Y 114.469,Z 481.402,A -85,B 0,C 180,E1 -26299.736,E2 -26299.736} C_VEL
LIN {X 0,Y 119.296,Z 489.622,A -85,B 0,C 180,E1 -26305.285,E2 -26305.285} C_VEL
LIN {X 0,Y 125.509,Z 496.315,A -85,B 0,C 180,E1 -26310.263,E2 -26310.263} C_VEL
LIN {X 0,Y 131.863,Z 500.956,A -85,B 0,C 180,E1 -26314.03,E2 -26314.03} C_VEL
LIN {X 0,Y 138.979,Z 504.654,A -85,B 0,C 180,E1 -26317.36,E2 -26317.36} C_VEL
LIN {X 0,Y 146.887,Z 507.478,A -85,B 0,C 180,E1 -26320.351,E2 -26320.351} C_VEL
LIN {X 0,Y 146.296,Z 507.714,A -85,B 0,C 180,E1 -26321.192,E2 -26321.192} C_VEL
LIN {X 0,Y 138.083,Z 507.166,A -85,B 0,C 180,E1 -26324.556,E2 -26324.556} C_VEL
LIN {X 0,Y 128.229,Z 505.485,A -85,B 0,C 180,E1 -26330.114,E2 -26330.114} C_VEL
LIN {X 0,Y 122.286,Z 503.508,A -85,B 0,C 180,E1 -26334.919,E2 -26334.919} C_VEL
LIN {X 0,Y 117.079,Z 500.378,A -85,B 0,C 180,E1 -26341.299,E2 -26341.299} C_VEL
LIN {X 0,Y 113.949,Z 496.29,A -85,B 0,C 180,E1 -26348.28,E2 -26348.28} C_VEL
LIN {X 0,Y 113.27,Z 491.12,A -85,B 0,C 180,E1 -26355.629,E2 -26355.629} C_VEL
LIN {X 0,Y 114.268,Z 486.341,A -85,B 0,C 180,E1 -26361.153,E2 -26361.153} C_VEL
LIN {X 0,Y 115.177,Z 483.26,A -85,B 0,C 180,E1 -26364.079,E2 -26364.079} C_VEL
LIN {X 0,Y 115.313,Z 480.786,A -85,B 0,C 180,E1 -26365.839,E2 -26365.839} C_VEL
LIN {X 0,Y 114.273,Z 471.615,A -85,B 0,C 180,E1 -26370.479,E2 -26370.479} C_VEL
LIN {X 0,Y 113.649,Z 460.826,A -85,B 0,C 180,E1 -26374.679,E2 -26374.679} C_VEL
LIN {X 0,Y 112.821,Z 455.798,A -85,B 0,C 180,E1 -26376.116,E2 -26376.116} C_VEL
LIN {X 0,Y 110.788,Z 442.707,A -85,B 0,C 180,E1 -26379.124,E2 -26379.124} C_VEL
LIN {X 0,Y 109.904,Z 431.269,A -85,B 0,C 180,E1 -26381.262,E2 -26381.262} C_VEL
LIN {X 0,Y 108.342,Z 428.346,A -85,B 0,C 180,E1 -26385.038,E2 -26385.038} C_VEL
LIN {X 0,Y 110.705,Z 415.431,A -85,B 0,C 180,E1 -26402.283,E2 -26402.283} C_VEL
LIN {X 0,Y 110.236,Z 413.25,A -85,B 0,C 180,E1 -26405.014,E2 -26405.014} C_VEL
LIN {X 0,Y 108.354,Z 406.989,A -85,B 0,C 180,E1 -26413.139,E2 -26413.139} C_VEL
LIN {X 0,Y 107.749,Z 407.063,A -85,B 0,C 180,E1 -26421.508,E2 -26421.508} C_VEL
LIN {X 0,Y 107.807,Z 407.056,A -85,B 0,C 180,E1 -26428.565,E2 -26428.565} C_VEL
LIN {X 0,Y 107.911,Z 407.041,A -85,B 0,C 180,E1 -26436.998,E2 -26436.998} C_VEL
LIN {X 0,Y 108.04,Z 407.024,A -85,B 0,C 180,E1 -26444.918,E2 -26444.918} C_VEL
LIN {X 0,Y 108.307,Z 406.992,A -85,B 0,C 180,E1 -26448.775,E2 -26448.775} C_VEL
LIN {X 0,Y 108.465,Z 406.973,A -85,B 0,C 180,E1 -26456.285,E2 -26456.285} C_VEL
LIN {X 0,Y 108.947,Z 406.907,A -85,B 0,C 180,E1 -26460,E2 -26460} C_VEL
LIN {X 0,Y 108.341,Z 406.984,A -85,B 0,C 180,E1 -26467.455,E2 -26467.455} C_VEL
LIN {X 0,Y 108.203,Z 407.007,A -85,B 0,C 180,E1 -26473.026,E2 -26473.026} C_VEL
LIN {X 0,Y 107.847,Z 407.04,A -85,B 0,C 180,E1 -26480.668,E2 -26480.668} C_VEL
LIN {X 0,Y 107.859,Z 407.046,A -85,B 0,C 180,E1 -26484.187,E2 -26484.187} C_VEL
LIN {X 0,Y 107.785,Z 407.057,A -85,B 0,C 180,E1 -26492.044,E2 -26492.044} C_VEL
LIN {X 0,Y 107.688,Z 407.066,A -85,B 0,C 180,E1 -26496.669,E2 -26496.669} C_VEL
LIN {X 0,Y 106.954,Z 407.161,A -85,B 0,C 180,E1 -26499.789,E2 -26499.789} C_VEL
LIN {X 0,Y 105.346,Z 407.361,A -85,B 0,C 180,E1 -26502.876,E2 -26502.876} C_VEL
LIN {X 0,Y 100.849,Z 407.915,A -85,B 0,C 180,E1 -26511.49,E2 -26511.49} C_VEL
LIN {X 0,Y 100.568,Z 407.942,A -85,B 0,C 180,E1 -26513.782,E2 -26513.782} C_VEL
LIN {X 0,Y 100.701,Z 407.94,A -85,B 0,C 180,E1 -26516.877,E2 -26516.877} C_VEL
LIN {X 0,Y 100.787,Z 407.93,A -85,B 0,C 180,E1 -26525.268,E2 -26525.268} C_VEL
LIN {X 0,Y 100.839,Z 407.918,A -85,B 0,C 180,E1 -26529.607,E2 -26529.607} C_VEL
LIN {X 0,Y 101.201,Z 407.872,A -85,B 0,C 180,E1 -26537.976,E2 -26537.976} C_VEL
LIN {X 0,Y 101.27,Z 407.871,A -85,B 0,C 180,E1 -26542.023,E2 -26542.023} C_VEL
LIN {X 0,Y 101.869,Z 407.797,A -85,B 0,C 180,E1 -26550.001,E2 -26550.001} C_VEL
LIN {X 0,Y 101.245,Z 407.874,A -85,B 0,C 180,E1 -26557.981,E2 -26557.981} C_VEL
LIN {X 0,Y 101.104,Z 407.883,A -85,B 0,C 180,E1 -26563.299,E2 -26563.299} C_VEL
LIN {X 0,Y 100.819,Z 407.921,A -85,B 0,C 180,E1 -26570.399,E2 -26570.399} C_VEL
LIN {X 0,Y 100.776,Z 407.931,A -85,B 0,C 180,E1 -26574.959,E2 -26574.959} C_VEL
LIN {X 0,Y 100.702,Z 407.94,A -85,B 0,C 180,E1 -26583.125,E2 -26583.125} C_VEL
LIN {X 0,Y 100.656,Z 407.942,A -85,B 0,C 180,E1 -26589.821,E2 -26589.821} C_VEL
LIN {X 0,Y 100.662,Z 407.941,A -85,B 0,C 180,E1 -26595.719,E2 -26595.719} C_VEL
LIN {X 0,Y 100.713,Z 407.94,A -85,B 0,C 180,E1 -26601.094,E2 -26601.094} C_VEL
LIN {X 0,Y 100.781,Z 407.917,A -85,B 0,C 180,E1 -26606.808,E2 -26606.808} C_VEL
LIN {X 0,Y 100.161,Z 408.008,A -85,B 0,C 180,E1 -26612.865,E2 -26612.865} C_VEL
LIN {X 0,Y 99.9,Z 408.201,A -85,B 0,C 180,E1 -26614.475,E2 -26614.475} C_VEL
LIN {X 0,Y 99.135,Z 412.473,A -85,B 0,C 180,E1 -26621.396,E2 -26621.396} C_VEL
LIN {X 0,Y 99.696,Z 418.987,A -85,B 0,C 180,E1 -26631.895,E2 -26631.895} C_VEL
LIN {X 0,Y 102.592,Z 422.99,A -85,B 0,C 180,E1 -26637.914,E2 -26637.914} C_VEL
LIN {X 0,Y 103.458,Z 428.716,A -85,B 0,C 180,E1 -26639.027,E2 -26639.027} C_VEL
LIN {X 0,Y 103.563,Z 440.559,A -85,B 0,C 180,E1 -26642.431,E2 -26642.431} C_VEL
LIN {X 0,Y 103.541,Z 449.843,A -85,B 0,C 180,E1 -26645.844,E2 -26645.844} C_VEL
LIN {X 0,Y 104.104,Z 460.534,A -85,B 0,C 180,E1 -26650.699,E2 -26650.699} C_VEL
LIN {X 0,Y 105.737,Z 471.148,A -85,B 0,C 180,E1 -26656.408,E2 -26656.408} C_VEL
LIN {X 0,Y 108.789,Z 479.952,A -85,B 0,C 180,E1 -26661.806,E2 -26661.806} C_VEL
LIN {X 0,Y 113.948,Z 488.606,A -85,B 0,C 180,E1 -26667.554,E2 -26667.554} C_VEL
LIN {X 0,Y 119.529,Z 494.644,A -85,B 0,C 180,E1 -26671.95,E2 -26671.95} C_VEL
LIN {X 0,Y 126.066,Z 499.776,A -85,B 0,C 180,E1 -26675.829,E2 -26675.829} C_VEL
LIN {X 0,Y 135.494,Z 504.839,A -85,B 0,C 180,E1 -26680.06,E2 -26680.06} C_VEL
LIN {X 0,Y 136.492,Z 505.273,A -85,B 0,C 180,E1 -26680.438,E2 -26680.438} C_VEL
LIN {X 0,Y 135.225,Z 505.388,A -85,B 0,C 180,E1 -26681.646,E2 -26681.646} C_VEL
LIN {X 0,Y 124.402,Z 503.325,A -85,B 0,C 180,E1 -26687.317,E2 -26687.317} C_VEL
LIN {X 0,Y 117.004,Z 500.694,A -85,B 0,C 180,E1 -26693.082,E2 -26693.082} C_VEL
LIN {X 0,Y 110.482,Z 496.213,A -85,B 0,C 180,E1 -26701.504,E2 -26701.504} C_VEL
LIN {X 0,Y 107.798,Z 491.583,A -85,B 0,C 180,E1 -26708.986,E2 -26708.986} C_VEL
LIN {X 0,Y 107.847,Z 484.875,A -85,B 0,C 180,E1 -26717.823,E2 -26717.823} C_VEL
LIN {X 0,Y 109.079,Z 480.374,A -85,B 0,C 180,E1 -26722.596,E2 -26722.596} C_VEL
LIN {X 0,Y 109.341,Z 479.129,A -85,B 0,C 180,E1 -26723.63,E2 -26723.63} C_VEL
LIN {X 0,Y 109.103,Z 476.137,A -85,B 0,C 180,E1 -26725.47,E2 -26725.47} C_VEL
LIN {X 0,Y 108.132,Z 467.909,A -85,B 0,C 180,E1 -26729.534,E2 -26729.534} C_VEL
LIN {X 0,Y 107.471,Z 458.614,A -85,B 0,C 180,E1 -26733.28,E2 -26733.28} C_VEL
LIN {X 0,Y 105.159,Z 446.945,A -85,B 0,C 180,E1 -26736.323,E2 -26736.323} C_VEL
LIN {X 0,Y 103.731,Z 434.313,A -85,B 0,C 180,E1 -26739.013,E2 -26739.013} C_VEL
LIN {X 0,Y 103.49,Z 430.936,A -85,B 0,C 180,E1 -26739.651,E2 -26739.651} C_VEL
LIN {X 0,Y 101.47,Z 427.626,A -85,B 0,C 180,E1 -26744.147,E2 -26744.147} C_VEL
LIN {X 0,Y 103.081,Z 416.248,A -85,B 0,C 180,E1 -26760.753,E2 -26760.753} C_VEL
LIN {X 0,Y 103.479,Z 414.687,A -85,B 0,C 180,E1 -26762.91,E2 -26762.91} C_VEL
LIN {X 0,Y 102.245,Z 410.755,A -85,B 0,C 180,E1 -26768.215,E2 -26768.215} C_VEL
LIN {X 0,Y 101.361,Z 407.861,A -85,B 0,C 180,E1 -26772.402,E2 -26772.402} C_VEL
LIN {X 0,Y 100.699,Z 407.941,A -85,B 0,C 180,E1 -26781.088,E2 -26781.088} C_VEL
LIN {X 0,Y 100.701,Z 407.936,A -85,B 0,C 180,E1 -26786.875,E2 -26786.875} C_VEL
LIN {X 0,Y 100.786,Z 407.924,A -85,B 0,C 180,E1 -26795.267,E2 -26795.267} C_VEL
LIN {X 0,Y 100.818,Z 407.927,A -85,B 0,C 180,E1 -26799.602,E2 -26799.602} C_VEL
LIN {X 0,Y 101.199,Z 407.879,A -85,B 0,C 180,E1 -26807.975,E2 -26807.975} C_VEL
LIN {X 0,Y 101.28,Z 407.862,A -85,B 0,C 180,E1 -26812.023,E2 -26812.023} C_VEL
LIN {X 0,Y 101.872,Z 407.788,A -85,B 0,C 180,E1 -26820,E2 -26820} C_VEL
LIN {X 0,Y 101.28,Z 407.862,A -85,B 0,C 180,E1 -26827.978,E2 -26827.978} C_VEL
LIN {X 0,Y 101.129,Z 407.888,A -85,B 0,C 180,E1 -26833.364,E2 -26833.364} C_VEL
LIN {X 0,Y 100.82,Z 407.925,A -85,B 0,C 180,E1 -26840.398,E2 -26840.398} C_VEL
LIN {X 0,Y 100.774,Z 407.925,A -85,B 0,C 180,E1 -26844.959,E2 -26844.959} C_VEL
LIN {X 0,Y 100.691,Z 407.936,A -85,B 0,C 180,E1 -26853.117,E2 -26853.117} C_VEL
LIN {X 0,Y 100.641,Z 407.948,A -85,B 0,C 180,E1 -26859.812,E2 -26859.812} C_VEL
LIN {X 0,Y 100.652,Z 407.946,A -85,B 0,C 180,E1 -26865.714,E2 -26865.714} C_VEL
LIN {X 0,Y 100.645,Z 407.94,A -85,B 0,C 180,E1 -26871.064,E2 -26871.064} C_VEL
LIN {X 0,Y 100.568,Z 407.942,A -85,B 0,C 180,E1 -26873.782,E2 -26873.782} C_VEL
LIN {X 0,Y 100.267,Z 407.995,A -85,B 0,C 180,E1 -26876.015,E2 -26876.015} C_VEL
LIN {X 0,Y 99.456,Z 408.093,A -85,B 0,C 180,E1 -26878.226,E2 -26878.226} C_VEL
LIN {X 0,Y 97.04,Z 408.396,A -85,B 0,C 180,E1 -26882.646,E2 -26882.646} C_VEL
LIN {X 0,Y 93.932,Z 408.779,A -85,B 0,C 180,E1 -26889.72,E2 -26889.72} C_VEL
LIN {X 0,Y 93.777,Z 408.801,A -85,B 0,C 180,E1 -26892.188,E2 -26892.188} C_VEL
LIN {X 0,Y 94.106,Z 408.754,A -85,B 0,C 180,E1 -26897.054,E2 -26897.054} C_VEL
LIN {X 0,Y 94.205,Z 408.75,A -85,B 0,C 180,E1 -26901.42,E2 -26901.42} C_VEL
LIN {X 0,Y 94.794,Z 408.678,A -85,B 0,C 180,E1 -26910.001,E2 -26910.001} C_VEL
LIN {X 0,Y 94.178,Z 408.754,A -85,B 0,C 180,E1 -26918.584,E2 -26918.584} C_VEL
LIN {X 0,Y 94.024,Z 408.765,A -85,B 0,C 180,E1 -26923.659,E2 -26923.659} C_VEL
LIN {X 0,Y 93.695,Z 408.807,A -85,B 0,C 180,E1 -26932.028,E2 -26932.028} C_VEL
LIN {X 0,Y 93.625,Z 408.822,A -85,B 0,C 180,E1 -26936.77,E2 -26936.77} C_VEL
LIN {X 0,Y 93.6,Z 408.825,A -85,B 0,C 180,E1 -26944.316,E2 -26944.316} C_VEL
LIN {X 0,Y 93.544,Z 408.832,A -85,B 0,C 180,E1 -26952.547,E2 -26952.547} C_VEL
LIN {X 0,Y 93.579,Z 408.824,A -85,B 0,C 180,E1 -26958.68,E2 -26958.68} C_VEL
LIN {X 0,Y 93.675,Z 408.806,A -85,B 0,C 180,E1 -26965.618,E2 -26965.618} C_VEL
LIN {X 0,Y 93.547,Z 408.825,A -85,B 0,C 180,E1 -26968.271,E2 -26968.271} C_VEL
LIN {X 0,Y 92.793,Z 408.925,A -85,B 0,C 180,E1 -26974.5,E2 -26974.5} C_VEL
LIN {X 0,Y 92.655,Z 408.947,A -85,B 0,C 180,E1 -26975.537,E2 -26975.537} C_VEL
LIN {X 0,Y 91.855,Z 414.053,A -85,B 0,C 180,E1 -26984.467,E2 -26984.467} C_VEL
LIN {X 0,Y 93.021,Z 419.294,A -85,B 0,C 180,E1 -26993.531,E2 -26993.531} C_VEL
LIN {X 0,Y 96.346,Z 423.307,A -85,B 0,C 180,E1 -26999.869,E2 -26999.869} C_VEL
LIN {X 0,Y 97.162,Z 428.947,A -85,B 0,C 180,E1 -27001.036,E2 -27001.036} C_VEL
LIN {X 0,Y 97.357,Z 440.555,A -85,B 0,C 180,E1 -27004.658,E2 -27004.658} C_VEL
LIN {X 0,Y 97.575,Z 451.891,A -85,B 0,C 180,E1 -27009.326,E2 -27009.326} C_VEL
LIN {X 0,Y 98.571,Z 462.281,A -85,B 0,C 180,E1 -27014.451,E2 -27014.451} C_VEL
LIN {X 0,Y 100.931,Z 472.453,A -85,B 0,C 180,E1 -27020.375,E2 -27020.375} C_VEL
LIN {X 0,Y 105.494,Z 482.489,A -85,B 0,C 180,E1 -27026.724,E2 -27026.724} C_VEL
LIN {X 0,Y 112.667,Z 491.704,A -85,B 0,C 180,E1 -27033.08,E2 -27033.08} C_VEL
LIN {X 0,Y 120.435,Z 498.241,A -85,B 0,C 180,E1 -27037.787,E2 -27037.787} C_VEL
LIN {X 0,Y 126.408,Z 501.992,A -85,B 0,C 180,E1 -27040.586,E2 -27040.586} C_VEL
LIN {X 0,Y 125.635,Z 502.181,A -85,B 0,C 180,E1 -27041.843,E2 -27041.843} C_VEL
LIN {X 0,Y 115.611,Z 499.242,A -85,B 0,C 180,E1 -27048.033,E2 -27048.033} C_VEL
LIN {X 0,Y 108.808,Z 495.838,A -85,B 0,C 180,E1 -27054.456,E2 -27054.456} C_VEL
LIN {X 0,Y 104.111,Z 491.599,A -85,B 0,C 180,E1 -27061.8,E2 -27061.8} C_VEL
LIN {X 0,Y 101.799,Z 484.909,A -85,B 0,C 180,E1 -27071.9,E2 -27071.9} C_VEL
LIN {X 0,Y 103.035,Z 477.673,A -85,B 0,C 180,E1 -27080.508,E2 -27080.508} C_VEL
LIN {X 0,Y 103.47,Z 475.939,A -85,B 0,C 180,E1 -27082.192,E2 -27082.192} C_VEL
LIN {X 0,Y 103.48,Z 474.596,A -85,B 0,C 180,E1 -27083.173,E2 -27083.173} C_VEL
LIN {X 0,Y 102.295,Z 466.167,A -85,B 0,C 180,E1 -27087.538,E2 -27087.538} C_VEL
LIN {X 0,Y 101.366,Z 456.549,A -85,B 0,C 180,E1 -27091.489,E2 -27091.489} C_VEL
LIN {X 0,Y 98.748,Z 443.711,A -85,B 0,C 180,E1 -27094.863,E2 -27094.863} C_VEL
LIN {X 0,Y 97.276,Z 430.586,A -85,B 0,C 180,E1 -27097.697,E2 -27097.697} C_VEL
LIN {X 0,Y 94.723,Z 427.047,A -85,B 0,C 180,E1 -27102.86,E2 -27102.86} C_VEL
LIN {X 0,Y 94.298,Z 419.973,A -85,B 0,C 180,E1 -27114.199,E2 -27114.199} C_VEL
LIN {X 0,Y 95.945,Z 415.767,A -85,B 0,C 180,E1 -27120.847,E2 -27120.847} C_VEL
LIN {X 0,Y 96.272,Z 414.187,A -85,B 0,C 180,E1 -27123.195,E2 -27123.195} C_VEL
LIN {X 0,Y 94.497,Z 408.781,A -85,B 0,C 180,E1 -27131.147,E2 -27131.147} C_VEL
LIN {X 0,Y 93.729,Z 408.804,A -85,B 0,C 180,E1 -27138.574,E2 -27138.574} C_VEL
LIN {X 0,Y 93.606,Z 408.817,A -85,B 0,C 180,E1 -27145.677,E2 -27145.677} C_VEL
LIN {X 0,Y 93.669,Z 408.809,A -85,B 0,C 180,E1 -27154.204,E2 -27154.204} C_VEL
LIN {X 0,Y 93.695,Z 408.814,A -85,B 0,C 180,E1 -27157.973,E2 -27157.973} C_VEL
LIN {X 0,Y 94.098,Z 408.764,A -85,B 0,C 180,E1 -27167.052,E2 -27167.052} C_VEL
LIN {X 0,Y 94.212,Z 408.742,A -85,B 0,C 180,E1 -27171.42,E2 -27171.42} C_VEL
LIN {X 0,Y 94.798,Z 408.669,A -85,B 0,C 180,E1 -27180,E2 -27180} C_VEL
LIN {X 0,Y 94.212,Z 408.741,A -85,B 0,C 180,E1 -27188.58,E2 -27188.58} C_VEL
LIN {X 0,Y 94.047,Z 408.769,A -85,B 0,C 180,E1 -27193.722,E2 -27193.722} C_VEL
LIN {X 0,Y 93.695,Z 408.813,A -85,B 0,C 180,E1 -27202.027,E2 -27202.027} C_VEL
LIN {X 0,Y 93.622,Z 408.816,A -85,B 0,C 180,E1 -27206.77,E2 -27206.77} C_VEL
LIN {X 0,Y 93.588,Z 408.819,A -85,B 0,C 180,E1 -27214.306,E2 -27214.306} C_VEL
LIN {X 0,Y 93.534,Z 408.826,A -85,B 0,C 180,E1 -27222.551,E2 -27222.551} C_VEL
LIN {X 0,Y 93.544,Z 408.831,A -85,B 0,C 180,E1 -27228.704,E2 -27228.704} C_VEL
LIN {X 0,Y 93.599,Z 408.826,A -85,B 0,C 180,E1 -27235.686,E2 -27235.686} C_VEL
LIN {X 0,Y 93.67,Z 408.818,A -85,B 0,C 180,E1 -27244.205,E2 -27244.205} C_VEL
LIN {X 0,Y 93.706,Z 408.805,A -85,B 0,C 180,E1 -27247.976,E2 -27247.976} C_VEL
LIN {X 0,Y 93.777,Z 408.801,A -85,B 0,C 180,E1 -27252.188,E2 -27252.188} C_VEL
LIN {X 0,Y 93.426,Z 408.866,A -85,B 0,C 180,E1 -27255.789,E2 -27255.789} C_VEL
LIN {X 0,Y 92.19,Z 409.026,A -85,B 0,C 180,E1 -27259.374,E2 -27259.374} C_VEL
LIN {X 0,Y 88.846,Z 409.425,A -85,B 0,C 180,E1 -27266.764,E2 -27266.764} C_VEL
LIN {X 0,Y 87.431,Z 409.583,A -85,B 0,C 180,E1 -27271.991,E2 -27271.991} C_VEL
LIN {X 0,Y 87.087,Z 409.637,A -85,B 0,C 180,E1 -27279.289,E2 -27279.289} C_VEL
LIN {X 0,Y 86.932,Z 409.65,A -85,B 0,C 180,E1 -27284.037,E2 -27284.037} C_VEL
LIN {X 0,Y 86.648,Z 409.69,A -85,B 0,C 180,E1 -27288.933,E2 -27288.933} C_VEL
LIN {X 0,Y 86.587,Z 409.699,A -85,B 0,C 180,E1 -27296.767,E2 -27296.767} C_VEL
LIN {X 0,Y 86.519,Z 409.706,A -85,B 0,C 180,E1 -27305.677,E2 -27305.677} C_VEL
LIN {X 0,Y 86.487,Z 409.712,A -85,B 0,C 180,E1 -27313,E2 -27313} C_VEL
LIN {X 0,Y 86.524,Z 409.705,A -85,B 0,C 180,E1 -27319.472,E2 -27319.472} C_VEL
LIN {X 0,Y 86.618,Z 409.686,A -85,B 0,C 180,E1 -27325.391,E2 -27325.391} C_VEL
LIN {X 0,Y 86.145,Z 409.755,A -85,B 0,C 180,E1 -27330.692,E2 -27330.692} C_VEL
LIN {X 0,Y 85.524,Z 409.831,A -85,B 0,C 180,E1 -27335.74,E2 -27335.74} C_VEL
LIN {X 0,Y 85.294,Z 410.07,A -85,B 0,C 180,E1 -27337.599,E2 -27337.599} C_VEL
LIN {X 0,Y 86.411,Z 419.566,A -85,B 0,C 180,E1 -27355.335,E2 -27355.335} C_VEL
LIN {X 0,Y 90.138,Z 423.532,A -85,B 0,C 180,E1 -27361.955,E2 -27361.955} C_VEL
LIN {X 0,Y 90.382,Z 423.818,A -85,B 0,C 180,E1 -27362.228,E2 -27362.228} C_VEL
LIN {X 0,Y 91.06,Z 428.668,A -85,B 0,C 180,E1 -27363.318,E2 -27363.318} C_VEL
LIN {X 0,Y 91.369,Z 440.169,A -85,B 0,C 180,E1 -27367.18,E2 -27367.18} C_VEL
LIN {X 0,Y 91.773,Z 451.559,A -85,B 0,C 180,E1 -27372.157,E2 -27372.157} C_VEL
LIN {X 0,Y 93.17,Z 461.783,A -85,B 0,C 180,E1 -27377.561,E2 -27377.561} C_VEL
LIN {X 0,Y 96.023,Z 472.097,A -85,B 0,C 180,E1 -27383.738,E2 -27383.738} C_VEL
LIN {X 0,Y 100.44,Z 480.826,A -85,B 0,C 180,E1 -27389.328,E2 -27389.328} C_VEL
LIN {X 0,Y 106.988,Z 489.396,A -85,B 0,C 180,E1 -27395.084,E2 -27395.084} C_VEL
LIN {X 0,Y 115.016,Z 496.437,A -85,B 0,C 180,E1 -27399.911,E2 -27399.911} C_VEL
LIN {X 0,Y 117.504,Z 498.243,A -85,B 0,C 180,E1 -27401.142,E2 -27401.142} C_VEL
LIN {X 0,Y 115.181,Z 497.686,A -85,B 0,C 180,E1 -27402.928,E2 -27402.928} C_VEL
LIN {X 0,Y 107.127,Z 494.311,A -85,B 0,C 180,E1 -27409,E2 -27409} C_VEL
LIN {X 0,Y 100.642,Z 489.773,A -85,B 0,C 180,E1 -27416.927,E2 -27416.927} C_VEL
LIN {X 0,Y 97.345,Z 485.149,A -85,B 0,C 180,E1 -27424.329,E2 -27424.329} C_VEL
LIN {X 0,Y 96.434,Z 479.07,A -85,B 0,C 180,E1 -27433.05,E2 -27433.05} C_VEL
LIN {X 0,Y 97.829,Z 472.29,A -85,B 0,C 180,E1 -27440.758,E2 -27440.758} C_VEL
LIN {X 0,Y 97.439,Z 469.136,A -85,B 0,C 180,E1 -27442.748,E2 -27442.748} C_VEL
LIN {X 0,Y 96.203,Z 460.901,A -85,B 0,C 180,E1 -27446.858,E2 -27446.858} C_VEL
LIN {X 0,Y 95.675,Z 456.033,A -85,B 0,C 180,E1 -27448.947,E2 -27448.947} C_VEL
LIN {X 0,Y 93.113,Z 444.603,A -85,B 0,C 180,E1 -27452.162,E2 -27452.162} C_VEL
LIN {X 0,Y 91.505,Z 432.932,A -85,B 0,C 180,E1 -27454.9,E2 -27454.9} C_VEL
LIN {X 0,Y 91.246,Z 430.327,A -85,B 0,C 180,E1 -27455.412,E2 -27455.412} C_VEL
LIN {X 0,Y 87.977,Z 426.379,A -85,B 0,C 180,E1 -27461.519,E2 -27461.519} C_VEL
LIN {X 0,Y 86.935,Z 420.74,A -85,B 0,C 180,E1 -27471.332,E2 -27471.332} C_VEL
LIN {X 0,Y 88.808,Z 415.209,A -85,B 0,C 180,E1 -27480.953,E2 -27480.953} C_VEL
LIN {X 0,Y 89.012,Z 413.602,A -85,B 0,C 180,E1 -27483.551,E2 -27483.551} C_VEL
LIN {X 0,Y 87.539,Z 409.583,A -85,B 0,C 180,E1 -27490.25,E2 -27490.25} C_VEL
LIN {X 0,Y 86.62,Z 409.693,A -85,B 0,C 180,E1 -27499.527,E2 -27499.527} C_VEL
LIN {X 0,Y 86.555,Z 409.695,A -85,B 0,C 180,E1 -27505.363,E2 -27505.363} C_VEL
LIN {X 0,Y 86.585,Z 409.693,A -85,B 0,C 180,E1 -27513.233,E2 -27513.233} C_VEL
LIN {X 0,Y 86.664,Z 409.686,A -85,B 0,C 180,E1 -27521.072,E2 -27521.072} C_VEL
LIN {X 0,Y 86.969,Z 409.651,A -85,B 0,C 180,E1 -27525.97,E2 -27525.97} C_VEL
LIN {X 0,Y 87.118,Z 409.626,A -85,B 0,C 180,E1 -27530.715,E2 -27530.715} C_VEL
LIN {X 0,Y 87.726,Z 409.549,A -85,B 0,C 180,E1 -27540,E2 -27540} C_VEL
LIN {X 0,Y 87.118,Z 409.625,A -85,B 0,C 180,E1 -27549.285,E2 -27549.285} C_VEL
LIN {X 0,Y 86.95,Z 409.653,A -85,B 0,C 180,E1 -27554.088,E2 -27554.088} C_VEL
LIN {X 0,Y 86.666,Z 409.685,A -85,B 0,C 180,E1 -27558.928,E2 -27558.928} C_VEL
LIN {X 0,Y 86.584,Z 409.693,A -85,B 0,C 180,E1 -27566.766,E2 -27566.766} C_VEL
LIN {X 0,Y 86.506,Z 409.704,A -85,B 0,C 180,E1 -27575.668,E2 -27575.668} C_VEL
LIN {X 0,Y 86.477,Z 409.705,A -85,B 0,C 180,E1 -27582.995,E2 -27582.995} C_VEL
LIN {X 0,Y 86.465,Z 409.711,A -85,B 0,C 180,E1 -27589.441,E2 -27589.441} C_VEL
LIN {X 0,Y 86.543,Z 409.705,A -85,B 0,C 180,E1 -27595.358,E2 -27595.358} C_VEL
LIN {X 0,Y 86.586,Z 409.699,A -85,B 0,C 180,E1 -27603.234,E2 -27603.234} C_VEL
LIN {X 0,Y 86.676,Z 409.687,A -85,B 0,C 180,E1 -27611.076,E2 -27611.076} C_VEL
LIN {X 0,Y 86.97,Z 409.645,A -85,B 0,C 180,E1 -27615.971,E2 -27615.971} C_VEL
LIN {X 0,Y 87.115,Z 409.634,A -85,B 0,C 180,E1 -27620.716,E2 -27620.716} C_VEL
LIN {X 0,Y 87.721,Z 409.559,A -85,B 0,C 180,E1 -27630.001,E2 -27630.001} C_VEL
LIN {X 0,Y 87.431,Z 409.583,A -85,B 0,C 180,E1 -27631.991,E2 -27631.991} C_VEL
LIN {X 0,Y 86.382,Z 409.721,A -85,B 0,C 180,E1 -27635.822,E2 -27635.822} C_VEL
LIN {X 0,Y 84.555,Z 409.952,A -85,B 0,C 180,E1 -27639.618,E2 -27639.618} C_VEL
LIN {X 0,Y 79.75,Z 410.544,A -85,B 0,C 180,E1 -27650.394,E2 -27650.394} C_VEL
LIN {X 0,Y 79.429,Z 410.575,A -85,B 0,C 180,E1 -27653.3,E2 -27653.3} C_VEL
LIN {X 0,Y 79.485,Z 410.581,A -85,B 0,C 180,E1 -27657.847,E2 -27657.847} C_VEL
LIN {X 0,Y 79.386,Z 410.593,A -85,B 0,C 180,E1 -27662.086,E2 -27662.086} C_VEL
LIN {X 0,Y 79.375,Z 410.589,A -85,B 0,C 180,E1 -27668.303,E2 -27668.303} C_VEL
LIN {X 0,Y 79.415,Z 410.589,A -85,B 0,C 180,E1 -27675.072,E2 -27675.072} C_VEL
LIN {X 0,Y 79.471,Z 410.585,A -85,B 0,C 180,E1 -27682.743,E2 -27682.743} C_VEL
LIN {X 0,Y 79.263,Z 410.602,A -85,B 0,C 180,E1 -27687.859,E2 -27687.859} C_VEL
LIN {X 0,Y 78.771,Z 410.67,A -85,B 0,C 180,E1 -27693.506,E2 -27693.506} C_VEL
LIN {X 0,Y 77.959,Z 410.93,A -85,B 0,C 180,E1 -27699.553,E2 -27699.553} C_VEL
LIN {X 0,Y 78.988,Z 418.415,A -85,B 0,C 180,E1 -27714.895,E2 -27714.895} C_VEL
LIN {X 0,Y 82.559,Z 422.539,A -85,B 0,C 180,E1 -27722.439,E2 -27722.439} C_VEL
LIN {X 0,Y 84.568,Z 424.056,A -85,B 0,C 180,E1 -27724.899,E2 -27724.899} C_VEL
LIN {X 0,Y 85.122,Z 427.975,A -85,B 0,C 180,E1 -27725.864,E2 -27725.864} C_VEL
LIN {X 0,Y 85.579,Z 439.744,A -85,B 0,C 180,E1 -27730.05,E2 -27730.05} C_VEL
LIN {X 0,Y 86.49,Z 452.014,A -85,B 0,C 180,E1 -27735.917,E2 -27735.917} C_VEL
LIN {X 0,Y 88.558,Z 463.077,A -85,B 0,C 180,E1 -27742.146,E2 -27742.146} C_VEL
LIN {X 0,Y 92.31,Z 473.078,A -85,B 0,C 180,E1 -27748.414,E2 -27748.414} C_VEL
LIN {X 0,Y 98.448,Z 483.028,A -85,B 0,C 180,E1 -27754.827,E2 -27754.827} C_VEL
LIN {X 0,Y 106.136,Z 491.24,A -85,B 0,C 180,E1 -27760.212,E2 -27760.212} C_VEL
LIN {X 0,Y 108.436,Z 493.238,A -85,B 0,C 180,E1 -27761.508,E2 -27761.508} C_VEL
LIN {X 0,Y 107.73,Z 493.209,A -85,B 0,C 180,E1 -27762.671,E2 -27762.671} C_VEL
LIN {X 0,Y 99.121,Z 488.646,A -85,B 0,C 180,E1 -27770.347,E2 -27770.347} C_VEL
LIN {X 0,Y 93.889,Z 483.747,A -85,B 0,C 180,E1 -27778.399,E2 -27778.399} C_VEL
LIN {X 0,Y 91.336,Z 477.87,A -85,B 0,C 180,E1 -27787.422,E2 -27787.422} C_VEL
LIN {X 0,Y 91.772,Z 470.787,A -85,B 0,C 180,E1 -27796.717,E2 -27796.717} C_VEL
LIN {X 0,Y 92.323,Z 468.672,A -85,B 0,C 180,E1 -27799.028,E2 -27799.028} C_VEL
LIN {X 0,Y 91.817,Z 465.182,A -85,B 0,C 180,E1 -27801.193,E2 -27801.193} C_VEL
LIN {X 0,Y 90.365,Z 456.251,A -85,B 0,C 180,E1 -27805.539,E2 -27805.539} C_VEL
LIN {X 0,Y 89.977,Z 453.619,A -85,B 0,C 180,E1 -27806.641,E2 -27806.641} C_VEL
LIN {X 0,Y 87.102,Z 441.624,A -85,B 0,C 180,E1 -27809.999,E2 -27809.999} C_VEL
LIN {X 0,Y 85.421,Z 429.942,A -85,B 0,C 180,E1 -27812.799,E2 -27812.799} C_VEL
LIN {X 0,Y 82.408,Z 427.111,A -85,B 0,C 180,E1 -27817.349,E2 -27817.349} C_VEL
LIN {X 0,Y 80.08,Z 422.803,A -85,B 0,C 180,E1 -27825.264,E2 -27825.264} C_VEL
LIN {X 0,Y 81.681,Z 414.606,A -85,B 0,C 180,E1 -27841.08,E2 -27841.08} C_VEL
LIN {X 0,Y 81.732,Z 412.969,A -85,B 0,C 180,E1 -27843.981,E2 -27843.981} C_VEL
LIN {X 0,Y 80.721,Z 410.43,A -85,B 0,C 180,E1 -27848.41,E2 -27848.41} C_VEL
LIN {X 0,Y 79.834,Z 410.537,A -85,B 0,C 180,E1 -27855.23,E2 -27855.23} C_VEL
LIN {X 0,Y 79.463,Z 410.585,A -85,B 0,C 180,E1 -27862.747,E2 -27862.747} C_VEL
LIN {X 0,Y 79.483,Z 410.581,A -85,B 0,C 180,E1 -27872.153,E2 -27872.153} C_VEL
LIN {X 0,Y 79.523,Z 410.579,A -85,B 0,C 180,E1 -27879.298,E2 -27879.298} C_VEL
LIN {X 0,Y 79.841,Z 410.538,A -85,B 0,C 180,E1 -27885.525,E2 -27885.525} C_VEL
LIN {X 0,Y 80.001,Z 410.514,A -85,B 0,C 180,E1 -27889.881,E2 -27889.881} C_VEL
LIN {X 0,Y 80.654,Z 410.43,A -85,B 0,C 180,E1 -27900,E2 -27900} C_VEL
LIN {X 0,Y 80,Z 410.515,A -85,B 0,C 180,E1 -27910.119,E2 -27910.119} C_VEL
LIN {X 0,Y 79.766,Z 410.544,A -85,B 0,C 180,E1 -27915.327,E2 -27915.327} C_VEL
LIN {X 0,Y 79.524,Z 410.579,A -85,B 0,C 180,E1 -27920.702,E2 -27920.702} C_VEL
LIN {X 0,Y 79.482,Z 410.581,A -85,B 0,C 180,E1 -27927.845,E2 -27927.845} C_VEL
LIN {X 0,Y 79.378,Z 410.595,A -85,B 0,C 180,E1 -27932.089,E2 -27932.089} C_VEL
LIN {X 0,Y 79.366,Z 410.599,A -85,B 0,C 180,E1 -27938.307,E2 -27938.307} C_VEL
LIN {X 0,Y 79.409,Z 410.59,A -85,B 0,C 180,E1 -27945.075,E2 -27945.075} C_VEL
LIN {X 0,Y 79.393,Z 410.589,A -85,B 0,C 180,E1 -27952.816,E2 -27952.816} C_VEL
LIN {X 0,Y 79.385,Z 410.593,A -85,B 0,C 180,E1 -27957.916,E2 -27957.916} C_VEL
LIN {X 0,Y 79.527,Z 410.578,A -85,B 0,C 180,E1 -27963.778,E2 -27963.778} C_VEL
LIN {X 0,Y 79.532,Z 410.571,A -85,B 0,C 180,E1 -27969.301,E2 -27969.301} C_VEL
LIN {X 0,Y 79.88,Z 410.53,A -85,B 0,C 180,E1 -27975.423,E2 -27975.423} C_VEL
LIN {X 0,Y 79.998,Z 410.518,A -85,B 0,C 180,E1 -27979.881,E2 -27979.881} C_VEL
LIN {X 0,Y 80.648,Z 410.44,A -85,B 0,C 180,E1 -27990.001,E2 -27990.001} C_VEL
LIN {X 0,Y 79.969,Z 410.522,A -85,B 0,C 180,E1 -28000.124,E2 -28000.124} C_VEL
LIN {X 0,Y 79.746,Z 410.549,A -85,B 0,C 180,E1 -28005.332,E2 -28005.332} C_VEL
LIN {X 0,Y 79.429,Z 410.575,A -85,B 0,C 180,E1 -28013.3,E2 -28013.3} C_VEL
LIN {X 0,Y 79.088,Z 410.633,A -85,B 0,C 180,E1 -28016.125,E2 -28016.125} C_VEL
LIN {X 0,Y 77.671,Z 410.807,A -85,B 0,C 180,E1 -28020.327,E2 -28020.327} C_VEL
LIN {X 0,Y 74.383,Z 411.218,A -85,B 0,C 180,E1 -28027.503,E2 -28027.503} C_VEL
LIN {X 0,Y 72.471,Z 411.457,A -85,B 0,C 180,E1 -28033.716,E2 -28033.716} C_VEL
LIN {X 0,Y 72.276,Z 411.473,A -85,B 0,C 180,E1 -28036.944,E2 -28036.944} C_VEL
LIN {X 0,Y 72.358,Z 411.472,A -85,B 0,C 180,E1 -28040.991,E2 -28040.991} C_VEL
LIN {X 0,Y 72.312,Z 411.471,A -85,B 0,C 180,E1 -28044.328,E2 -28044.328} C_VEL
LIN {X 0,Y 71.814,Z 411.539,A -85,B 0,C 180,E1 -28051.739,E2 -28051.739} C_VEL
LIN {X 0,Y 70.701,Z 411.725,A -85,B 0,C 180,E1 -28061.902,E2 -28061.902} C_VEL
LIN {X 0,Y 72.464,Z 418.592,A -85,B 0,C 180,E1 -28077.22,E2 -28077.22} C_VEL
LIN {X 0,Y 76.646,Z 422.726,A -85,B 0,C 180,E1 -28085.261,E2 -28085.261} C_VEL
LIN {X 0,Y 79.106,Z 424.568,A -85,B 0,C 180,E1 -28088.108,E2 -28088.108} C_VEL
LIN {X 0,Y 79.446,Z 427.621,A -85,B 0,C 180,E1 -28088.976,E2 -28088.976} C_VEL
LIN {X 0,Y 80.061,Z 437.42,A -85,B 0,C 180,E1 -28092.677,E2 -28092.677} C_VEL
LIN {X 0,Y 81.193,Z 449.923,A -85,B 0,C 180,E1 -28098.81,E2 -28098.81} C_VEL
LIN {X 0,Y 82.904,Z 458.509,A -85,B 0,C 180,E1 -28103.745,E2 -28103.745} C_VEL
LIN {X 0,Y 87.559,Z 470.813,A -85,B 0,C 180,E1 -28111.448,E2 -28111.448} C_VEL
LIN {X 0,Y 93.136,Z 479.734,A -85,B 0,C 180,E1 -28117.134,E2 -28117.134} C_VEL
LIN {X 0,Y 99.829,Z 487.371,A -85,B 0,C 180,E1 -28121.975,E2 -28121.975} C_VEL
LIN {X 0,Y 98.305,Z 486.953,A -85,B 0,C 180,E1 -28124.362,E2 -28124.362} C_VEL
LIN {X 0,Y 90.259,Z 480.908,A -85,B 0,C 180,E1 -28134.268,E2 -28134.268} C_VEL
LIN {X 0,Y 86.36,Z 473.34,A -85,B 0,C 180,E1 -28145.989,E2 -28145.989} C_VEL
LIN {X 0,Y 86.866,Z 465.64,A -85,B 0,C 180,E1 -28156.139,E2 -28156.139} C_VEL
LIN {X 0,Y 87.033,Z 464.851,A -85,B 0,C 180,E1 -28157.049,E2 -28157.049} C_VEL
LIN {X 0,Y 86.312,Z 461.001,A -85,B 0,C 180,E1 -28159.441,E2 -28159.441} C_VEL
LIN {X 0,Y 84.854,Z 452.839,A -85,B 0,C 180,E1 -28163.401,E2 -28163.401} C_VEL
LIN {X 0,Y 81.715,Z 440.731,A -85,B 0,C 180,E1 -28166.918,E2 -28166.918} C_VEL
LIN {X 0,Y 79.937,Z 429.626,A -85,B 0,C 180,E1 -28169.684,E2 -28169.684} C_VEL
LIN {X 0,Y 75.96,Z 426.338,A -85,B 0,C 180,E1 -28175.308,E2 -28175.308} C_VEL
LIN {X 0,Y 73.021,Z 421.191,A -85,B 0,C 180,E1 -28185.748,E2 -28185.748} C_VEL
LIN {X 0,Y 74.614,Z 413.596,A -85,B 0,C 180,E1 -28202.035,E2 -28202.035} C_VEL
LIN {X 0,Y 74.038,Z 411.414,A -85,B 0,C 180,E1 -28206.209,E2 -28206.209} C_VEL
LIN {X 0,Y 72.55,Z 411.439,A -85,B 0,C 180,E1 -28217.305,E2 -28217.305} C_VEL
LIN {X 0,Y 72.344,Z 411.467,A -85,B 0,C 180,E1 -28224.346,E2 -28224.346} C_VEL
LIN {X 0,Y 72.391,Z 411.467,A -85,B 0,C 180,E1 -28230.96,E2 -28230.96} C_VEL
LIN {X 0,Y 72.399,Z 411.465,A -85,B 0,C 180,E1 -28237.152,E2 -28237.152} C_VEL
LIN {X 0,Y 72.757,Z 411.419,A -85,B 0,C 180,E1 -28245.003,E2 -28245.003} C_VEL
LIN {X 0,Y 72.885,Z 411.404,A -85,B 0,C 180,E1 -28248.881,E2 -28248.881} C_VEL
LIN {X 0,Y 73.581,Z 411.311,A -85,B 0,C 180,E1 -28260,E2 -28260} C_VEL
LIN {X 0,Y 72.885,Z 411.404,A -85,B 0,C 180,E1 -28271.119,E2 -28271.119} C_VEL
LIN {X 0,Y 72.586,Z 411.435,A -85,B 0,C 180,E1 -28276.886,E2 -28276.886} C_VEL
LIN {X 0,Y 72.4,Z 411.465,A -85,B 0,C 180,E1 -28282.848,E2 -28282.848} C_VEL
LIN {X 0,Y 72.376,Z 411.469,A -85,B 0,C 180,E1 -28289.083,E2 -28289.083} C_VEL
LIN {X 0,Y 72.294,Z 411.473,A -85,B 0,C 180,E1 -28295.682,E2 -28295.682} C_VEL
LIN {X 0,Y 72.259,Z 411.475,A -85,B 0,C 180,E1 -28302.908,E2 -28302.908} C_VEL
LIN {X 0,Y 72.301,Z 411.47,A -85,B 0,C 180,E1 -28311.046,E2 -28311.046} C_VEL
LIN {X 0,Y 72.3,Z 411.477,A -85,B 0,C 180,E1 -28314.323,E2 -28314.323} C_VEL
LIN {X 0,Y 72.375,Z 411.462,A -85,B 0,C 180,E1 -28320.954,E2 -28320.954} C_VEL
LIN {X 0,Y 72.405,Z 411.46,A -85,B 0,C 180,E1 -28327.155,E2 -28327.155} C_VEL
LIN {X 0,Y 72.783,Z 411.416,A -85,B 0,C 180,E1 -28334.93,E2 -28334.93} C_VEL
LIN {X 0,Y 72.893,Z 411.4,A -85,B 0,C 180,E1 -28338.883,E2 -28338.883} C_VEL
LIN {X 0,Y 73.573,Z 411.321,A -85,B 0,C 180,E1 -28350.001,E2 -28350.001} C_VEL
LIN {X 0,Y 72.86,Z 411.404,A -85,B 0,C 180,E1 -28361.124,E2 -28361.124} C_VEL
LIN {X 0,Y 72.575,Z 411.445,A -85,B 0,C 180,E1 -28366.89,E2 -28366.89} C_VEL
LIN {X 0,Y 72.383,Z 411.461,A -85,B 0,C 180,E1 -28373.027,E2 -28373.027} C_VEL
LIN {X 0,Y 72.378,Z 411.462,A -85,B 0,C 180,E1 -28379.083,E2 -28379.083} C_VEL
LIN {X 0,Y 72.302,Z 411.477,A -85,B 0,C 180,E1 -28385.679,E2 -28385.679} C_VEL
LIN {X 0,Y 72.265,Z 411.484,A -85,B 0,C 180,E1 -28392.906,E2 -28392.906} C_VEL
LIN {X 0,Y 72.276,Z 411.473,A -85,B 0,C 180,E1 -28396.944,E2 -28396.944} C_VEL
LIN {X 0,Y 72.004,Z 411.515,A -85,B 0,C 180,E1 -28400.035,E2 -28400.035} C_VEL
LIN {X 0,Y 70.478,Z 411.712,A -85,B 0,C 180,E1 -28404.62,E2 -28404.62} C_VEL
LIN {X 0,Y 68.26,Z 411.988,A -85,B 0,C 180,E1 -28409.203,E2 -28409.203} C_VEL
LIN {X 0,Y 64.072,Z 412.503,A -85,B 0,C 180,E1 -28419.414,E2 -28419.414} C_VEL
LIN {X 0,Y 63.551,Z 412.56,A -85,B 0,C 180,E1 -28423.116,E2 -28423.116} C_VEL
LIN {X 0,Y 63.558,Z 412.798,A -85,B 0,C 180,E1 -28425.594,E2 -28425.594} C_VEL
LIN {X 0,Y 66.088,Z 418.695,A -85,B 0,C 180,E1 -28440,E2 -28440} C_VEL
LIN {X 0,Y 71.108,Z 422.985,A -85,B 0,C 180,E1 -28448.745,E2 -28448.745} C_VEL
LIN {X 0,Y 73.988,Z 424.793,A -85,B 0,C 180,E1 -28451.819,E2 -28451.819} C_VEL
LIN {X 0,Y 74.754,Z 434.85,A -85,B 0,C 180,E1 -28455.648,E2 -28455.648} C_VEL
LIN {X 0,Y 76.097,Z 446.824,A -85,B 0,C 180,E1 -28461.68,E2 -28461.68} C_VEL
LIN {X 0,Y 78.66,Z 457.486,A -85,B 0,C 180,E1 -28467.974,E2 -28467.974} C_VEL
LIN {X 0,Y 83.151,Z 468.309,A -85,B 0,C 180,E1 -28474.786,E2 -28474.786} C_VEL
LIN {X 0,Y 90.279,Z 478.942,A -85,B 0,C 180,E1 -28481.43,E2 -28481.43} C_VEL
LIN {X 0,Y 92.586,Z 481.69,A -85,B 0,C 180,E1 -28483.092,E2 -28483.092} C_VEL
LIN {X 0,Y 88.839,Z 479.153,A -85,B 0,C 180,E1 -28487.744,E2 -28487.744} C_VEL
LIN {X 0,Y 83.297,Z 472.988,A -85,B 0,C 180,E1 -28497.536,E2 -28497.536} C_VEL
LIN {X 0,Y 81.432,Z 464.781,A -85,B 0,C 180,E1 -28509.804,E2 -28509.804} C_VEL
LIN {X 0,Y 81.982,Z 460.491,A -85,B 0,C 180,E1 -28515.096,E2 -28515.096} C_VEL
LIN {X 0,Y 80.247,Z 452.727,A -85,B 0,C 180,E1 -28519.273,E2 -28519.273} C_VEL
LIN {X 0,Y 79.635,Z 450.172,A -85,B 0,C 180,E1 -28520.326,E2 -28520.326} C_VEL
LIN {X 0,Y 76.323,Z 438.114,A -85,B 0,C 180,E1 -28523.816,E2 -28523.816} C_VEL
LIN {X 0,Y 74.74,Z 429.269,A -85,B 0,C 180,E1 -28526.124,E2 -28526.124} C_VEL
LIN {X 0,Y 70.311,Z 426.076,A -85,B 0,C 180,E1 -28531.703,E2 -28531.703} C_VEL
LIN {X 0,Y 66.455,Z 421.268,A -85,B 0,C 180,E1 -28542.21,E2 -28542.21} C_VEL
LIN {X 0,Y 67.357,Z 413.294,A -85,B 0,C 180,E1 -28561.445,E2 -28561.445} C_VEL
LIN {X 0,Y 67.272,Z 412.106,A -85,B 0,C 180,E1 -28564.129,E2 -28564.129} C_VEL
LIN {X 0,Y 66.002,Z 412.265,A -85,B 0,C 180,E1 -28571.809,E2 -28571.809} C_VEL
LIN {X 0,Y 65.389,Z 412.338,A -85,B 0,C 180,E1 -28579.844,E2 -28579.844} C_VEL
LIN {X 0,Y 65.26,Z 412.356,A -85,B 0,C 180,E1 -28589.487,E2 -28589.487} C_VEL
LIN {X 0,Y 65.248,Z 412.348,A -85,B 0,C 180,E1 -28594.479,E2 -28594.479} C_VEL
LIN {X 0,Y 65.651,Z 412.301,A -85,B 0,C 180,E1 -28604.459,E2 -28604.459} C_VEL
LIN {X 0,Y 65.783,Z 412.291,A -85,B 0,C 180,E1 -28607.662,E2 -28607.662} C_VEL
LIN {X 0,Y 66.505,Z 412.192,A -85,B 0,C 180,E1 -28620,E2 -28620} C_VEL
LIN {X 0,Y 65.783,Z 412.291,A -85,B 0,C 180,E1 -28632.338,E2 -28632.338} C_VEL
LIN {X 0,Y 65.39,Z 412.334,A -85,B 0,C 180,E1 -28638.81,E2 -28638.81} C_VEL
LIN {X 0,Y 65.24,Z 412.349,A -85,B 0,C 180,E1 -28645.525,E2 -28645.525} C_VEL
LIN {X 0,Y 65.195,Z 412.358,A -85,B 0,C 180,E1 -28652.616,E2 -28652.616} C_VEL
LIN {X 0,Y 65.19,Z 412.36,A -85,B 0,C 180,E1 -28661.006,E2 -28661.006} C_VEL
LIN {X 0,Y 65.211,Z 412.356,A -85,B 0,C 180,E1 -28669.713,E2 -28669.713} C_VEL
LIN {X 0,Y 65.255,Z 412.348,A -85,B 0,C 180,E1 -28679.498,E2 -28679.498} C_VEL
LIN {X 0,Y 65.245,Z 412.358,A -85,B 0,C 180,E1 -28684.479,E2 -28684.479} C_VEL
LIN {X 0,Y 65.672,Z 412.303,A -85,B 0,C 180,E1 -28694.398,E2 -28694.398} C_VEL
LIN {X 0,Y 65.798,Z 412.28,A -85,B 0,C 180,E1 -28697.666,E2 -28697.666} C_VEL
LIN {X 0,Y 66.496,Z 412.203,A -85,B 0,C 180,E1 -28710.001,E2 -28710.001} C_VEL
LIN {X 0,Y 65.757,Z 412.285,A -85,B 0,C 180,E1 -28722.344,E2 -28722.344} C_VEL
LIN {X 0,Y 65.382,Z 412.339,A -85,B 0,C 180,E1 -28728.814,E2 -28728.814} C_VEL
LIN {X 0,Y 65.241,Z 412.359,A -85,B 0,C 180,E1 -28735.526,E2 -28735.526} C_VEL
LIN {X 0,Y 65.2,Z 412.361,A -85,B 0,C 180,E1 -28742.614,E2 -28742.614} C_VEL
LIN {X 0,Y 65.196,Z 412.361,A -85,B 0,C 180,E1 -28751.011,E2 -28751.011} C_VEL
LIN {X 0,Y 65.254,Z 412.354,A -85,B 0,C 180,E1 -28759.743,E2 -28759.743} C_VEL
LIN {X 0,Y 64.968,Z 412.38,A -85,B 0,C 180,E1 -28767.256,E2 -28767.256} C_VEL
LIN {X 0,Y 64.834,Z 412.41,A -85,B 0,C 180,E1 -28770.137,E2 -28770.137} C_VEL
LIN {X 0,Y 64.377,Z 412.46,A -85,B 0,C 180,E1 -28774.108,E2 -28774.108} C_VEL
LIN {X 0,Y 63.551,Z 412.56,A -85,B 0,C 180,E1 -28783.116,E2 -28783.116} C_VEL
LIN {X 0,Y 63.152,Z 413.36,A -85,B 0,C 180,E1 -28787.104,E2 -28787.104} C_VEL
LIN {X 0,Y 61.996,Z 415.68,A -85,B 0,C 180,E1 -28793.588,E2 -28793.588} C_VEL
LIN {X 0,Y 61.769,Z 419.978,A -85,B 0,C 180,E1 -28805.658,E2 -28805.658} C_VEL
LIN {X 0,Y 63.839,Z 421.883,A -85,B 0,C 180,E1 -28810.267,E2 -28810.267} C_VEL
LIN {X 0,Y 69.083,Z 425.236,A -85,B 0,C 180,E1 -28816.309,E2 -28816.309} C_VEL
LIN {X 0,Y 69.991,Z 433.64,A -85,B 0,C 180,E1 -28819.81,E2 -28819.81} C_VEL
LIN {X 0,Y 72.145,Z 446.991,A -85,B 0,C 180,E1 -28826.958,E2 -28826.958} C_VEL
LIN {X 0,Y 75.657,Z 458.295,A -85,B 0,C 180,E1 -28833.873,E2 -28833.873} C_VEL
LIN {X 0,Y 82.231,Z 470.507,A -85,B 0,C 180,E1 -28841.48,E2 -28841.48} C_VEL
LIN {X 0,Y 84.701,Z 474.013,A -85,B 0,C 180,E1 -28843.577,E2 -28843.577} C_VEL
LIN {X 0,Y 85.053,Z 474.777,A -85,B 0,C 180,E1 -28845.029,E2 -28845.029} C_VEL
LIN {X 0,Y 78.356,Z 466.927,A -85,B 0,C 180,E1 -28857.44,E2 -28857.44} C_VEL
LIN {X 0,Y 76.908,Z 459.518,A -85,B 0,C 180,E1 -28868.559,E2 -28868.559} C_VEL
LIN {X 0,Y 77.176,Z 456.851,A -85,B 0,C 180,E1 -28872.074,E2 -28872.074} C_VEL
LIN {X 0,Y 76.464,Z 453.716,A -85,B 0,C 180,E1 -28873.993,E2 -28873.993} C_VEL
LIN {X 0,Y 75.392,Z 449.366,A -85,B 0,C 180,E1 -28876.142,E2 -28876.142} C_VEL
LIN {X 0,Y 71.566,Z 436.479,A -85,B 0,C 180,E1 -28879.888,E2 -28879.888} C_VEL
LIN {X 0,Y 70.022,Z 428.933,A -85,B 0,C 180,E1 -28881.922,E2 -28881.922} C_VEL
LIN {X 0,Y 65.394,Z 426.11,A -85,B 0,C 180,E1 -28886.918,E2 -28886.918} C_VEL
LIN {X 0,Y 60.655,Z 421.802,A -85,B 0,C 180,E1 -28896.652,E2 -28896.652} C_VEL
LIN {X 0,Y 60.081,Z 412.999,A -85,B 0,C 180,E1 -28920.896,E2 -28920.896} C_VEL
LIN {X 0,Y 60.015,Z 413.009,A -85,B 0,C 180,E1 -28924.943,E2 -28924.943} C_VEL
LIN {X 0,Y 58.483,Z 413.192,A -85,B 0,C 180,E1 -28936.138,E2 -28936.138} C_VEL
LIN {X 0,Y 58.174,Z 413.234,A -85,B 0,C 180,E1 -28947.742,E2 -28947.742} C_VEL
LIN {X 0,Y 58.158,Z 413.24,A -85,B 0,C 180,E1 -28951.094,E2 -28951.094} C_VEL
LIN {X 0,Y 58.537,Z 413.185,A -85,B 0,C 180,E1 -28963.835,E2 -28963.835} C_VEL
LIN {X 0,Y 58.826,Z 413.151,A -85,B 0,C 180,E1 -28973.138,E2 -28973.138} C_VEL
LIN {X 0,Y 59.397,Z 413.077,A -85,B 0,C 180,E1 -28980,E2 -28980} C_VEL
LIN {X 0,Y 58.825,Z 413.151,A -85,B 0,C 180,E1 -28986.862,E2 -28986.862} C_VEL
LIN {X 0,Y 58.537,Z 413.185,A -85,B 0,C 180,E1 -28996.166,E2 -28996.166} C_VEL
LIN {X 0,Y 58.151,Z 413.24,A -85,B 0,C 180,E1 -29008.91,E2 -29008.91} C_VEL
LIN {X 0,Y 58.157,Z 413.236,A -85,B 0,C 180,E1 -29012.232,E2 -29012.232} C_VEL
LIN {X 0,Y 58.034,Z 413.254,A -85,B 0,C 180,E1 -29017.266,E2 -29017.266} C_VEL
LIN {X 0,Y 58.02,Z 413.258,A -85,B 0,C 180,E1 -29026.617,E2 -29026.617} C_VEL
LIN {X 0,Y 58.037,Z 413.248,A -85,B 0,C 180,E1 -29032.739,E2 -29032.739} C_VEL
LIN {X 0,Y 58.159,Z 413.236,A -85,B 0,C 180,E1 -29037.767,E2 -29037.767} C_VEL
LIN {X 0,Y 58.153,Z 413.233,A -85,B 0,C 180,E1 -29041.093,E2 -29041.093} C_VEL
LIN {X 0,Y 58.555,Z 413.191,A -85,B 0,C 180,E1 -29053.78,E2 -29053.78} C_VEL
LIN {X 0,Y 58.676,Z 413.167,A -85,B 0,C 180,E1 -29056.141,E2 -29056.141} C_VEL
LIN {X 0,Y 58.825,Z 413.155,A -85,B 0,C 180,E1 -29063.14,E2 -29063.14} C_VEL
LIN {X 0,Y 59.387,Z 413.088,A -85,B 0,C 180,E1 -29070.001,E2 -29070.001} C_VEL
LIN {X 0,Y 58.802,Z 413.158,A -85,B 0,C 180,E1 -29076.866,E2 -29076.866} C_VEL
LIN {X 0,Y 58.518,Z 413.195,A -85,B 0,C 180,E1 -29086.095,E2 -29086.095} C_VEL
LIN {X 0,Y 58.152,Z 413.233,A -85,B 0,C 180,E1 -29098.911,E2 -29098.911} C_VEL
LIN {X 0,Y 58.161,Z 413.236,A -85,B 0,C 180,E1 -29102.235,E2 -29102.235} C_VEL
LIN {X 0,Y 58.057,Z 413.253,A -85,B 0,C 180,E1 -29113.421,E2 -29113.421} C_VEL
LIN {X 0,Y 58.07,Z 413.243,A -85,B 0,C 180,E1 -29116.567,E2 -29116.567} C_VEL
LIN {X 0,Y 57.985,Z 413.261,A -85,B 0,C 180,E1 -29122.698,E2 -29122.698} C_VEL
LIN {X 0,Y 57.857,Z 413.271,A -85,B 0,C 180,E1 -29128.247,E2 -29128.247} C_VEL
LIN {X 0,Y 57.641,Z 413.305,A -85,B 0,C 180,E1 -29130.81,E2 -29130.81} C_VEL
LIN {X 0,Y 56.494,Z 413.433,A -85,B 0,C 180,E1 -29142.945,E2 -29142.945} C_VEL
LIN {X 0,Y 56.625,Z 413.464,A -85,B 0,C 180,E1 -29149.166,E2 -29149.166} C_VEL
LIN {X 0,Y 59.919,Z 418.779,A -85,B 0,C 180,E1 -29163.362,E2 -29163.362} C_VEL
LIN {X 0,Y 63.839,Z 421.883,A -85,B 0,C 180,E1 -29170.267,E2 -29170.267} C_VEL
LIN {X 0,Y 65.267,Z 423.454,A -85,B 0,C 180,E1 -29173.278,E2 -29173.278} C_VEL
LIN {X 0,Y 65.793,Z 425.298,A -85,B 0,C 180,E1 -29176.414,E2 -29176.414} C_VEL
LIN {X 0,Y 65.81,Z 428.224,A -85,B 0,C 180,E1 -29180.499,E2 -29180.499} C_VEL
LIN {X 0,Y 65.803,Z 431.911,A -85,B 0,C 180,E1 -29184.136,E2 -29184.136} C_VEL
LIN {X 0,Y 66.016,Z 434.128,A -85,B 0,C 180,E1 -29185.57,E2 -29185.57} C_VEL
LIN {X 0,Y 68.05,Z 444.201,A -85,B 0,C 180,E1 -29191.09,E2 -29191.09} C_VEL
LIN {X 0,Y 72.847,Z 457.221,A -85,B 0,C 180,E1 -29199.192,E2 -29199.192} C_VEL
LIN {X 0,Y 78.885,Z 467.692,A -85,B 0,C 180,E1 -29205.458,E2 -29205.458} C_VEL
LIN {X 0,Y 77.924,Z 466.749,A -85,B 0,C 180,E1 -29207.43,E2 -29207.43} C_VEL
LIN {X 0,Y 73.238,Z 459.01,A -85,B 0,C 180,E1 -29219.729,E2 -29219.729} C_VEL
LIN {X 0,Y 72.775,Z 452.603,A -85,B 0,C 180,E1 -29229.124,E2 -29229.124} C_VEL
LIN {X 0,Y 71.399,Z 447.876,A -85,B 0,C 180,E1 -29231.7,E2 -29231.7} C_VEL
LIN {X 0,Y 67.339,Z 435.411,A -85,B 0,C 180,E1 -29235.261,E2 -29235.261} C_VEL
LIN {X 0,Y 65.754,Z 428.568,A -85,B 0,C 180,E1 -29237.124,E2 -29237.124} C_VEL
LIN {X 0,Y 59.644,Z 425.153,A -85,B 0,C 180,E1 -29243.232,E2 -29243.232} C_VEL
LIN {X 0,Y 54.239,Z 420.921,A -85,B 0,C 180,E1 -29253.713,E2 -29253.713} C_VEL
LIN {X 0,Y 52.234,Z 413.981,A -85,B 0,C 180,E1 -29275.929,E2 -29275.929} C_VEL
LIN {X 0,Y 53.082,Z 413.871,A -85,B 0,C 180,E1 -29281.977,E2 -29281.977} C_VEL
LIN {X 0,Y 52.506,Z 413.942,A -85,B 0,C 180,E1 -29286.573,E2 -29286.573} C_VEL
LIN {X 0,Y 51.356,Z 414.078,A -85,B 0,C 180,E1 -29296.823,E2 -29296.823} C_VEL
LIN {X 0,Y 51.082,Z 414.113,A -85,B 0,C 180,E1 -29306.61,E2 -29306.61} C_VEL
LIN {X 0,Y 51.03,Z 414.121,A -85,B 0,C 180,E1 -29315.596,E2 -29315.596} C_VEL
LIN {X 0,Y 51.482,Z 414.064,A -85,B 0,C 180,E1 -29324.156,E2 -29324.156} C_VEL
LIN {X 0,Y 51.701,Z 414.036,A -85,B 0,C 180,E1 -29332.187,E2 -29332.187} C_VEL
LIN {X 0,Y 52.282,Z 413.963,A -85,B 0,C 180,E1 -29340,E2 -29340} C_VEL
LIN {X 0,Y 51.701,Z 414.036,A -85,B 0,C 180,E1 -29347.813,E2 -29347.813} C_VEL
LIN {X 0,Y 51.403,Z 414.072,A -85,B 0,C 180,E1 -29356.856,E2 -29356.856} C_VEL
LIN {X 0,Y 51.026,Z 414.121,A -85,B 0,C 180,E1 -29364.407,E2 -29364.407} C_VEL
LIN {X 0,Y 51.005,Z 414.122,A -85,B 0,C 180,E1 -29374.237,E2 -29374.237} C_VEL
LIN {X 0,Y 50.986,Z 414.125,A -85,B 0,C 180,E1 -29383.568,E2 -29383.568} C_VEL
LIN {X 0,Y 51.032,Z 414.129,A -85,B 0,C 180,E1 -29395.722,E2 -29395.722} C_VEL
LIN {X 0,Y 51.032,Z 414.126,A -85,B 0,C 180,E1 -29405.598,E2 -29405.598} C_VEL
LIN {X 0,Y 51.505,Z 414.068,A -85,B 0,C 180,E1 -29414.164,E2 -29414.164} C_VEL
LIN {X 0,Y 51.705,Z 414.044,A -85,B 0,C 180,E1 -29422.189,E2 -29422.189} C_VEL
LIN {X 0,Y 52.27,Z 413.975,A -85,B 0,C 180,E1 -29430.001,E2 -29430.001} C_VEL
LIN {X 0,Y 51.678,Z 414.047,A -85,B 0,C 180,E1 -29437.818,E2 -29437.818} C_VEL
LIN {X 0,Y 51.388,Z 414.084,A -85,B 0,C 180,E1 -29446.793,E2 -29446.793} C_VEL
LIN {X 0,Y 51.025,Z 414.127,A -85,B 0,C 180,E1 -29454.409,E2 -29454.409} C_VEL
LIN {X 0,Y 51.034,Z 414.128,A -85,B 0,C 180,E1 -29464.281,E2 -29464.281} C_VEL
LIN {X 0,Y 51.025,Z 414.129,A -85,B 0,C 180,E1 -29473.528,E2 -29473.528} C_VEL
LIN {X 0,Y 51.034,Z 414.119,A -85,B 0,C 180,E1 -29476.483,E2 -29476.483} C_VEL
LIN {X 0,Y 50.795,Z 414.145,A -85,B 0,C 180,E1 -29486.396,E2 -29486.396} C_VEL
LIN {X 0,Y 49.981,Z 414.252,A -85,B 0,C 180,E1 -29495.049,E2 -29495.049} C_VEL
LIN {X 0,Y 50.061,Z 414.313,A -85,B 0,C 180,E1 -29514.461,E2 -29514.461} C_VEL
LIN {X 0,Y 54.023,Z 418.811,A -85,B 0,C 180,E1 -29527.475,E2 -29527.475} C_VEL
LIN {X 0,Y 64.892,Z 425.686,A -85,B 0,C 180,E1 -29541.648,E2 -29541.648} C_VEL
LIN {X 0,Y 66.016,Z 434.128,A -85,B 0,C 180,E1 -29545.57,E2 -29545.57} C_VEL
LIN {X 0,Y 66.442,Z 438.788,A -85,B 0,C 180,E1 -29548.69,E2 -29548.69} C_VEL
LIN {X 0,Y 66.966,Z 445.333,A -85,B 0,C 180,E1 -29555.095,E2 -29555.095} C_VEL
LIN {X 0,Y 68.611,Z 451.574,A -85,B 0,C 180,E1 -29561.556,E2 -29561.556} C_VEL
LIN {X 0,Y 70.554,Z 455.778,A -85,B 0,C 180,E1 -29564.642,E2 -29564.642} C_VEL
LIN {X 0,Y 72.632,Z 459.342,A -85,B 0,C 180,E1 -29566.736,E2 -29566.736} C_VEL
LIN {X 0,Y 72.898,Z 459.841,A -85,B 0,C 180,E1 -29567.555,E2 -29567.555} C_VEL
LIN {X 0,Y 68.929,Z 451.395,A -85,B 0,C 180,E1 -29581.147,E2 -29581.147} C_VEL
LIN {X 0,Y 68.761,Z 449.215,A -85,B 0,C 180,E1 -29584.365,E2 -29584.365} C_VEL
LIN {X 0,Y 68.61,Z 447.939,A -85,B 0,C 180,E1 -29585.81,E2 -29585.81} C_VEL
LIN {X 0,Y 67.601,Z 445.058,A -85,B 0,C 180,E1 -29587.053,E2 -29587.053} C_VEL
LIN {X 0,Y 63.289,Z 432.123,A -85,B 0,C 180,E1 -29590.539,E2 -29590.539} C_VEL
LIN {X 0,Y 62.195,Z 428.172,A -85,B 0,C 180,E1 -29591.615,E2 -29591.615} C_VEL
LIN {X 0,Y 54.189,Z 424.165,A -85,B 0,C 180,E1 -29598.781,E2 -29598.781} C_VEL
LIN {X 0,Y 48.025,Z 420.003,A -85,B 0,C 180,E1 -29609.998,E2 -29609.998} C_VEL
LIN {X 0,Y 44.945,Z 414.887,A -85,B 0,C 180,E1 -29628.222,E2 -29628.222} C_VEL
LIN {X 0,Y 45.337,Z 414.836,A -85,B 0,C 180,E1 -29637.712,E2 -29637.712} C_VEL
LIN {X 0,Y 45.025,Z 414.869,A -85,B 0,C 180,E1 -29648.698,E2 -29648.698} C_VEL
LIN {X 0,Y 43.991,Z 415.001,A -85,B 0,C 180,E1 -29663.014,E2 -29663.014} C_VEL
LIN {X 0,Y 43.86,Z 415.019,A -85,B 0,C 180,E1 -29671.268,E2 -29671.268} C_VEL
LIN {X 0,Y 44.257,Z 414.962,A -85,B 0,C 180,E1 -29682.319,E2 -29682.319} C_VEL
LIN {X 0,Y 44.553,Z 414.926,A -85,B 0,C 180,E1 -29690.924,E2 -29690.924} C_VEL
LIN {X 0,Y 45.158,Z 414.85,A -85,B 0,C 180,E1 -29700,E2 -29700} C_VEL
LIN {X 0,Y 44.552,Z 414.926,A -85,B 0,C 180,E1 -29709.076,E2 -29709.076} C_VEL
LIN {X 0,Y 44.193,Z 414.972,A -85,B 0,C 180,E1 -29718.546,E2 -29718.546} C_VEL
LIN {X 0,Y 43.843,Z 415.021,A -85,B 0,C 180,E1 -29728.744,E2 -29728.744} C_VEL
LIN {X 0,Y 43.796,Z 415.027,A -85,B 0,C 180,E1 -29739.933,E2 -29739.933} C_VEL
LIN {X 0,Y 43.844,Z 415.016,A -85,B 0,C 180,E1 -29753.271,E2 -29753.271} C_VEL
LIN {X 0,Y 43.847,Z 415.014,A -85,B 0,C 180,E1 -29761.261,E2 -29761.261} C_VEL
LIN {X 0,Y 44.264,Z 414.971,A -85,B 0,C 180,E1 -29772.297,E2 -29772.297} C_VEL
LIN {X 0,Y 44.561,Z 414.934,A -85,B 0,C 180,E1 -29780.927,E2 -29780.927} C_VEL
LIN {X 0,Y 45.144,Z 414.862,A -85,B 0,C 180,E1 -29790.002,E2 -29790.002} C_VEL
LIN {X 0,Y 44.531,Z 414.938,A -85,B 0,C 180,E1 -29799.082,E2 -29799.082} C_VEL
LIN {X 0,Y 44.154,Z 414.982,A -85,B 0,C 180,E1 -29808.565,E2 -29808.565} C_VEL
LIN {X 0,Y 43.845,Z 415.015,A -85,B 0,C 180,E1 -29818.745,E2 -29818.745} C_VEL
LIN {X 0,Y 43.827,Z 415.017,A -85,B 0,C 180,E1 -29829.901,E2 -29829.901} C_VEL
LIN {X 0,Y 43.754,Z 415.032,A -85,B 0,C 180,E1 -29840.021,E2 -29840.021} C_VEL
LIN {X 0,Y 43.702,Z 415.034,A -85,B 0,C 180,E1 -29843.525,E2 -29843.525} C_VEL
LIN {X 0,Y 43.156,Z 415.109,A -85,B 0,C 180,E1 -29850.754,E2 -29850.754} C_VEL
LIN {X 0,Y 42.469,Z 415.189,A -85,B 0,C 180,E1 -29860.672,E2 -29860.672} C_VEL
LIN {X 0,Y 44.164,Z 415.095,A -85,B 0,C 180,E1 -29881.14,E2 -29881.14} C_VEL
LIN {X 0,Y 51.565,Z 420.712,A -85,B 0,C 180,E1 -29897.431,E2 -29897.431} C_VEL
LIN {X 0,Y 58.47,Z 424.405,A -85,B 0,C 180,E1 -29904.878,E2 -29904.878} C_VEL
LIN {X 0,Y 61.22,Z 425.868,A -85,B 0,C 180,E1 -29907.567,E2 -29907.567} C_VEL
LIN {X 0,Y 63.163,Z 435.997,A -85,B 0,C 180,E1 -29912.849,E2 -29912.849} C_VEL
LIN {X 0,Y 65.917,Z 445.176,A -85,B 0,C 180,E1 -29918.194,E2 -29918.194} C_VEL
LIN {X 0,Y 70.554,Z 455.778,A -85,B 0,C 180,E1 -29924.642,E2 -29924.642} C_VEL
LIN {X 0,Y 70.817,Z 456.435,A -85,B 0,C 180,E1 -29925.615,E2 -29925.615} C_VEL
LIN {X 0,Y 70.493,Z 456.224,A -85,B 0,C 180,E1 -29927.667,E2 -29927.667} C_VEL
LIN {X 0,Y 69.421,Z 454.598,A -85,B 0,C 180,E1 -29930.285,E2 -29930.285} C_VEL
LIN {X 0,Y 65.595,Z 446.707,A -85,B 0,C 180,E1 -29937.828,E2 -29937.828} C_VEL
LIN {X 0,Y 65.264,Z 445.309,A -85,B 0,C 180,E1 -29939.697,E2 -29939.697} C_VEL
LIN {X 0,Y 65.15,Z 444.316,A -85,B 0,C 180,E1 -29941.216,E2 -29941.216} C_VEL
LIN {X 0,Y 60.779,Z 432.331,A -85,B 0,C 180,E1 -29944.301,E2 -29944.301} C_VEL
LIN {X 0,Y 59.293,Z 427.825,A -85,B 0,C 180,E1 -29945.489,E2 -29945.489} C_VEL
LIN {X 0,Y 52.287,Z 424.712,A -85,B 0,C 180,E1 -29950.202,E2 -29950.202} C_VEL
LIN {X 0,Y 44.072,Z 420.382,A -85,B 0,C 180,E1 -29960.822,E2 -29960.822} C_VEL
LIN {X 0,Y 38.565,Z 415.677,A -85,B 0,C 180,E1 -29979.173,E2 -29979.173} C_VEL
LIN {X 0,Y 37.846,Z 415.763,A -85,B 0,C 180,E1 -29991.8,E2 -29991.8} C_VEL
LIN {X 0,Y 37.93,Z 415.76,A -85,B 0,C 180,E1 -30003.768,E2 -30003.768} C_VEL
LIN {X 0,Y 37.514,Z 415.808,A -85,B 0,C 180,E1 -30011.465,E2 -30011.465} C_VEL
LIN {X 0,Y 36.817,Z 415.889,A -85,B 0,C 180,E1 -30025.064,E2 -30025.064} C_VEL
LIN {X 0,Y 37.081,Z 415.857,A -85,B 0,C 180,E1 -30041.372,E2 -30041.372} C_VEL
LIN {X 0,Y 37.35,Z 415.826,A -85,B 0,C 180,E1 -30049.154,E2 -30049.154} C_VEL
LIN {X 0,Y 38.017,Z 415.739,A -85,B 0,C 180,E1 -30060,E2 -30060} C_VEL
LIN {X 0,Y 37.35,Z 415.826,A -85,B 0,C 180,E1 -30070.846,E2 -30070.846} C_VEL
LIN {X 0,Y 37.079,Z 415.857,A -85,B 0,C 180,E1 -30078.619,E2 -30078.619} C_VEL
LIN {X 0,Y 36.712,Z 415.902,A -85,B 0,C 180,E1 -30095.052,E2 -30095.052} C_VEL
LIN {X 0,Y 36.719,Z 415.906,A -85,B 0,C 180,E1 -30100.042,E2 -30100.042} C_VEL
LIN {X 0,Y 36.725,Z 415.902,A -85,B 0,C 180,E1 -30109.949,E2 -30109.949} C_VEL
LIN {X 0,Y 36.725,Z 415.909,A -85,B 0,C 180,E1 -30114.966,E2 -30114.966} C_VEL
LIN {X 0,Y 37.085,Z 415.861,A -85,B 0,C 180,E1 -30131.364,E2 -30131.364} C_VEL
LIN {X 0,Y 37.357,Z 415.824,A -85,B 0,C 180,E1 -30139.158,E2 -30139.158} C_VEL
LIN {X 0,Y 38.002,Z 415.752,A -85,B 0,C 180,E1 -30150.002,E2 -30150.002} C_VEL
LIN {X 0,Y 37.328,Z 415.828,A -85,B 0,C 180,E1 -30160.854,E2 -30160.854} C_VEL
LIN {X 0,Y 37.056,Z 415.865,A -85,B 0,C 180,E1 -30168.505,E2 -30168.505} C_VEL
LIN {X 0,Y 36.731,Z 415.908,A -85,B 0,C 180,E1 -30185.033,E2 -30185.033} C_VEL
LIN {X 0,Y 36.738,Z 415.9,A -85,B 0,C 180,E1 -30190.075,E2 -30190.075} C_VEL
LIN {X 0,Y 36.712,Z 415.907,A -85,B 0,C 180,E1 -30199.977,E2 -30199.977} C_VEL
LIN {X 0,Y 36.457,Z 415.934,A -85,B 0,C 180,E1 -30204.667,E2 -30204.667} C_VEL
LIN {X 0,Y 35.534,Z 416.053,A -85,B 0,C 180,E1 -30216.698,E2 -30216.698} C_VEL
LIN {X 0,Y 38.894,Z 415.655,A -85,B 0,C 180,E1 -30249.097,E2 -30249.097} C_VEL
LIN {X 0,Y 45.427,Z 419.827,A -85,B 0,C 180,E1 -30261.829,E2 -30261.829} C_VEL
LIN {X 0,Y 54.547,Z 424.347,A -85,B 0,C 180,E1 -30271.023,E2 -30271.023} C_VEL
LIN {X 0,Y 58.711,Z 426.572,A -85,B 0,C 180,E1 -30274.653,E2 -30274.653} C_VEL
LIN {X 0,Y 62.155,Z 439.262,A -85,B 0,C 180,E1 -30281.628,E2 -30281.628} C_VEL
LIN {X 0,Y 66.519,Z 449.47,A -85,B 0,C 180,E1 -30287.696,E2 -30287.696} C_VEL
LIN {X 0,Y 67.694,Z 451.604,A -85,B 0,C 180,E1 -30288.941,E2 -30288.941} C_VEL
LIN {X 0,Y 66.211,Z 448.64,A -85,B 0,C 180,E1 -30294.28,E2 -30294.28} C_VEL
LIN {X 0,Y 65.264,Z 445.309,A -85,B 0,C 180,E1 -30299.697,E2 -30299.697} C_VEL
LIN {X 0,Y 64.799,Z 444.1,A -85,B 0,C 180,E1 -30300.333,E2 -30300.333} C_VEL
LIN {X 0,Y 63.484,Z 441.604,A -85,B 0,C 180,E1 -30299.852,E2 -30299.852} C_VEL
LIN {X 0,Y 60.897,Z 436.814,A -85,B 0,C 180,E1 -30297.209,E2 -30297.209} C_VEL
LIN {X 0,Y 60.067,Z 434.845,A -85,B 0,C 180,E1 -30297.064,E2 -30297.064} C_VEL
LIN {X 0,Y 57.446,Z 427.465,A -85,B 0,C 180,E1 -30298.69,E2 -30298.69} C_VEL
LIN {X 0,Y 47.936,Z 423.587,A -85,B 0,C 180,E1 -30303.905,E2 -30303.905} C_VEL
LIN {X 0,Y 38.878,Z 419.38,A -85,B 0,C 180,E1 -30314.265,E2 -30314.265} C_VEL
LIN {X 0,Y 33.632,Z 416.281,A -85,B 0,C 180,E1 -30327.332,E2 -30327.332} C_VEL
LIN {X 0,Y 30.653,Z 416.565,A -85,B 0,C 180,E1 -30357.291,E2 -30357.291} C_VEL
LIN {X 0,Y 30.082,Z 416.617,A -85,B 0,C 180,E1 -30375.503,E2 -30375.503} C_VEL
LIN {X 0,Y 29.583,Z 416.665,A -85,B 0,C 180,E1 -30391.632,E2 -30391.632} C_VEL
LIN {X 0,Y 29.892,Z 416.636,A -85,B 0,C 180,E1 -30400.118,E2 -30400.118} C_VEL
LIN {X 0,Y 30.128,Z 416.615,A -85,B 0,C 180,E1 -30406.51,E2 -30406.51} C_VEL
LIN {X 0,Y 30.836,Z 416.544,A -85,B 0,C 180,E1 -30420,E2 -30420} C_VEL
LIN {X 0,Y 30.127,Z 416.615,A -85,B 0,C 180,E1 -30433.491,E2 -30433.491} C_VEL
LIN {X 0,Y 29.889,Z 416.636,A -85,B 0,C 180,E1 -30439.861,E2 -30439.861} C_VEL
LIN {X 0,Y 29.503,Z 416.672,A -85,B 0,C 180,E1 -30448.453,E2 -30448.453} C_VEL
LIN {X 0,Y 29.54,Z 416.669,A -85,B 0,C 180,E1 -30465.542,E2 -30465.542} C_VEL
LIN {X 0,Y 29.512,Z 416.671,A -85,B 0,C 180,E1 -30481.56,E2 -30481.56} C_VEL
LIN {X 0,Y 29.893,Z 416.635,A -85,B 0,C 180,E1 -30490.122,E2 -30490.122} C_VEL
LIN {X 0,Y 30.133,Z 416.611,A -85,B 0,C 180,E1 -30496.515,E2 -30496.515} C_VEL
LIN {X 0,Y 30.819,Z 416.551,A -85,B 0,C 180,E1 -30510.003,E2 -30510.003} C_VEL
LIN {X 0,Y 30.106,Z 416.613,A -85,B 0,C 180,E1 -30523.502,E2 -30523.502} C_VEL
LIN {X 0,Y 29.865,Z 416.637,A -85,B 0,C 180,E1 -30529.725,E2 -30529.725} C_VEL
LIN {X 0,Y 29.5,Z 416.671,A -85,B 0,C 180,E1 -30538.459,E2 -30538.459} C_VEL
LIN {X 0,Y 29.54,Z 416.668,A -85,B 0,C 180,E1 -30555.544,E2 -30555.544} C_VEL
LIN {X 0,Y 28.698,Z 416.747,A -85,B 0,C 180,E1 -30570.673,E2 -30570.673} C_VEL
LIN {X 0,Y 28.44,Z 416.771,A -85,B 0,C 180,E1 -30591.312,E2 -30591.312} C_VEL
LIN {X 0,Y 34.646,Z 416.193,A -85,B 0,C 180,E1 -30619.247,E2 -30619.247} C_VEL
LIN {X 0,Y 45.005,Z 421.389,A -85,B 0,C 180,E1 -30633.131,E2 -30633.131} C_VEL
LIN {X 0,Y 51.319,Z 424.216,A -85,B 0,C 180,E1 -30638.044,E2 -30638.044} C_VEL
LIN {X 0,Y 57.043,Z 426.915,A -85,B 0,C 180,E1 -30642.359,E2 -30642.359} C_VEL
LIN {X 0,Y 60.342,Z 436.828,A -85,B 0,C 180,E1 -30647.665,E2 -30647.665} C_VEL
LIN {X 0,Y 63.156,Z 442.993,A -85,B 0,C 180,E1 -30651.166,E2 -30651.166} C_VEL
LIN {X 0,Y 62.321,Z 440.507,A -85,B 0,C 180,E1 -30655.676,E2 -30655.676} C_VEL
LIN {X 0,Y 60.067,Z 434.845,A -85,B 0,C 180,E1 -30657.064,E2 -30657.064} C_VEL
LIN {X 0,Y 58.209,Z 431.549,A -85,B 0,C 180,E1 -30657.719,E2 -30657.719} C_VEL
LIN {X 0,Y 54.06,Z 427.488,A -85,B 0,C 180,E1 -30658.311,E2 -30658.311} C_VEL
LIN {X 0,Y 49.028,Z 424.388,A -85,B 0,C 180,E1 -30658.813,E2 -30658.813} C_VEL
LIN {X 0,Y 41.584,Z 421.313,A -85,B 0,C 180,E1 -30660.39,E2 -30660.39} C_VEL
LIN {X 0,Y 36.276,Z 419.176,A -85,B 0,C 180,E1 -30663.618,E2 -30663.618} C_VEL
LIN {X 0,Y 34.699,Z 418.501,A -85,B 0,C 180,E1 -30665.407,E2 -30665.407} C_VEL
LIN {X 0,Y 30.3,Z 416.599,A -85,B 0,C 180,E1 -30673.143,E2 -30673.143} C_VEL
LIN {X 0,Y 23.514,Z 417.043,A -85,B 0,C 180,E1 -30716.277,E2 -30716.277} C_VEL
LIN {X 0,Y 22.937,Z 417.061,A -85,B 0,C 180,E1 -30727.789,E2 -30727.789} C_VEL
LIN {X 0,Y 22.523,Z 417.074,A -85,B 0,C 180,E1 -30741.386,E2 -30741.386} C_VEL
LIN {X 0,Y 22.844,Z 417.064,A -85,B 0,C 180,E1 -30762.083,E2 -30762.083} C_VEL
LIN {X 0,Y 23.604,Z 417.041,A -85,B 0,C 180,E1 -30780,E2 -30780} C_VEL
LIN {X 0,Y 22.841,Z 417.064,A -85,B 0,C 180,E1 -30797.921,E2 -30797.921} C_VEL
LIN {X 0,Y 22.195,Z 417.085,A -85,B 0,C 180,E1 -30819.294,E2 -30819.294} C_VEL
LIN {X 0,Y 22.198,Z 417.085,A -85,B 0,C 180,E1 -30830.717,E2 -30830.717} C_VEL
LIN {X 0,Y 22.846,Z 417.064,A -85,B 0,C 180,E1 -30852.087,E2 -30852.087} C_VEL
LIN {X 0,Y 23.588,Z 417.041,A -85,B 0,C 180,E1 -30870.003,E2 -30870.003} C_VEL
LIN {X 0,Y 22.813,Z 417.065,A -85,B 0,C 180,E1 -30887.947,E2 -30887.947} C_VEL
LIN {X 0,Y 22.197,Z 417.084,A -85,B 0,C 180,E1 -30909.295,E2 -30909.295} C_VEL
LIN {X 0,Y 21.888,Z 417.094,A -85,B 0,C 180,E1 -30920.045,E2 -30920.045} C_VEL
LIN {X 0,Y 21.102,Z 417.119,A -85,B 0,C 180,E1 -30940.546,E2 -30940.546} C_VEL
LIN {X 0,Y 24.906,Z 417,A -85,B 0,C 180,E1 -30976.39,E2 -30976.39} C_VEL
LIN {X 0,Y 31.574,Z 416.572,A -85,B 0,C 180,E1 -30991.406,E2 -30991.406} C_VEL
LIN {X 0,Y 48.97,Z 423.984,A -85,B 0,C 180,E1 -31005.856,E2 -31005.856} C_VEL
LIN {X 0,Y 55.237,Z 426.544,A -85,B 0,C 180,E1 -31009.765,E2 -31009.765} C_VEL
LIN {X 0,Y 56.558,Z 427.123,A -85,B 0,C 180,E1 -31011.587,E2 -31011.587} C_VEL
LIN {X 0,Y 44.596,Z 422.572,A -85,B 0,C 180,E1 -31016.271,E2 -31016.271} C_VEL
LIN {X 0,Y 34.699,Z 418.501,A -85,B 0,C 180,E1 -31025.407,E2 -31025.407} C_VEL
LIN {X 0,Y 30.236,Z 417.286,A -85,B 0,C 180,E1 -31031.855,E2 -31031.855} C_VEL
LIN {X 0,Y 25.782,Z 417.013,A -85,B 0,C 180,E1 -31039.885,E2 -31039.885} C_VEL
LIN {X 0,Y 18.054,Z 417.178,A -85,B 0,C 180,E1 -31064.505,E2 -31064.505} C_VEL
LIN {X 0,Y 15.178,Z 417.178,A -85,B 0,C 180,E1 -31090.766,E2 -31090.766} C_VEL
LIN {X 0,Y 15.368,Z 417.178,A -85,B 0,C 180,E1 -31116.142,E2 -31116.142} C_VEL
LIN {X 0,Y 16.276,Z 417.178,A -85,B 0,C 180,E1 -31140,E2 -31140} C_VEL
LIN {X 0,Y 15.286,Z 417.178,A -85,B 0,C 180,E1 -31163.153,E2 -31163.153} C_VEL
LIN {X 0,Y 15.106,Z 417.178,A -85,B 0,C 180,E1 -31167.726,E2 -31167.726} C_VEL
LIN {X 0,Y 15.111,Z 417.178,A -85,B 0,C 180,E1 -31202.289,E2 -31202.289} C_VEL
LIN {X 0,Y 15.29,Z 417.178,A -85,B 0,C 180,E1 -31206.829,E2 -31206.829} C_VEL
LIN {X 0,Y 16.257,Z 417.178,A -85,B 0,C 180,E1 -31230.005,E2 -31230.005} C_VEL
LIN {X 0,Y 15.259,Z 417.178,A -85,B 0,C 180,E1 -31252.898,E2 -31252.898} C_VEL
LIN {X 0,Y 14.797,Z 417.178,A -85,B 0,C 180,E1 -31276.536,E2 -31276.536} C_VEL
LIN {X 0,Y 14.18,Z 417.178,A -85,B 0,C 180,E1 -31312.467,E2 -31312.467} C_VEL
LIN {X 0,Y 23.379,Z 417.048,A -85,B 0,C 180,E1 -31356.957,E2 -31356.957} C_VEL
LIN {X 0,Y 29.846,Z 416.771,A -85,B 0,C 180,E1 -31364.944,E2 -31364.944} C_VEL
LIN {X 0,Y 36.854,Z 419.534,A -85,B 0,C 180,E1 -31369.712,E2 -31369.712} C_VEL
LIN {X 0,Y 36.386,Z 419.373,A -85,B 0,C 180,E1 -31370.589,E2 -31370.589} C_VEL
LIN {X 0,Y 29.134,Z 416.708,A -85,B 0,C 180,E1 -31377.125,E2 -31377.125} C_VEL
LIN {X 0,Y 21.718,Z 417.099,A -85,B 0,C 180,E1 -31391.115,E2 -31391.115} C_VEL
LIN {X 0,Y 16.298,Z 417.178,A -85,B 0,C 180,E1 -31435.539,E2 -31435.539} C_VEL
LIN {X 0,Y 15.178,Z 417.178,A -85,B 0,C 180,E1 -31450.766,E2 -31450.766} C_VEL
LIN {X 0,Y 14.415,Z 417.178,A -85,B 0,C 180,E1 -31458.823,E2 -31458.823} C_VEL
LIN {X 0,Y 12.242,Z 417.178,A -85,B 0,C 180,E1 -31472.172,E2 -31472.172} C_VEL
LIN {X 0,Y 10.193,Z 417.178,A -85,B 0,C 180,E1 -31485.365,E2 -31485.365} C_VEL
LIN {X 0,Y 8.505,Z 417.178,A -85,B 0,C 180,E1 -31502.851,E2 -31502.851} C_VEL
LIN {X 0,Y 7.78,Z 417.178,A -85,B 0,C 180,E1 -31525.427,E2 -31525.427} C_VEL
LIN {X 0,Y 7.782,Z 417.178,A -85,B 0,C 180,E1 -31564.572,E2 -31564.572} C_VEL
LIN {X 0,Y 8.685,Z 417.178,A -85,B 0,C 180,E1 -31590.009,E2 -31590.009} C_VEL
LIN {X 0,Y 7.856,Z 417.178,A -85,B 0,C 180,E1 -31616.538,E2 -31616.538} C_VEL
LIN {X 0,Y 7.207,Z 417.178,A -85,B 0,C 180,E1 -31679.999,E2 -31679.999} C_VEL
LIN {X 0,Y 18.015,Z 417.178,A -85,B 0,C 180,E1 -31731.282,E2 -31731.282} C_VEL
LIN {X 0,Y 17.199,Z 417.178,A -85,B 0,C 180,E1 -31734.81,E2 -31734.81} C_VEL
LIN {X 0,Y 10.003,Z 417.178,A -85,B 0,C 180,E1 -31769.992,E2 -31769.992} C_VEL
LIN {X 0,Y 8.303,Z 417.178,A -85,B 0,C 180,E1 -31802.171,E2 -31802.171} C_VEL
LIN {X 0,Y 7.992,Z 417.178,A -85,B 0,C 180,E1 -31831.548,E2 -31831.548} C_VEL
LIN {X 0,Y 8.707,Z 417.178,A -85,B 0,C 180,E1 -31860.001,E2 -31860.001} C_VEL
LIN {X 0,Y 8.505,Z 417.178,A -85,B 0,C 180,E1 -31862.851,E2 -31862.851} C_VEL
LIN {X 0,Y 7.911,Z 419.178,A -85,B 0,C 180,E1 -31876.221,E2 -31876.221} C_VEL
LIN {X 0,Y 7.911,Z 600,A -85,B 0,C 180,E1 -31876.221,E2 -31876.221} C_VEL
LIN {X 0,Y 7.911,Z 600,A -85,B 0,C 180,E1 -31876.221,E2 -31876.221}

QRS_NEXT_CUT()

QRS_NEXT()
QRS_HOME()

END
